(* IEC 61131-3 sources: Intern_HiERN_Testplattform_Hoplyt/Intern_HiERN_Testplattform_PLC, 10 files *)

(* ---- GlobalVariables.gvl ---- *)
VAR_GLOBAL
	MFC_INSTANCE : MFC_BHFF;

	MFC_CONTROLLER: FB_Bronkhorst_FFDevice_RTU;

	CORIFLOW_INSTANCE : BH_DeviceSingle;
	CORIFLOW_CONTROLLER: FB_Bronkhorst_SingleDevice;

	ELPRESS_INSTANCE : BH_DeviceSingle;
	ELPRESS_CONTROLLER: FB_Bronkhorst_SingleDevice;

	TESTCASE: TESTCASE;

	(* HW *)
	Read_SV_flow : REAL;
	Read_AV_flow : REAL;
	Read_unit_flow : STRING;
	Read_alarm_info_flow : SINT;

	Read_SV_p_up : REAL;
	Read_AV_p_up : REAL;
	Read_unit_p_up : STRING;
	Read_alarm_info_p_up : SINT;

	Read_SV_p_down : REAL;
	Read_AV_p_down : REAL;
	Read_unit_p_down : STRING;
	Read_alarm_info_p_down : SINT;

	Read_temperature: REAL;
	Read_density: REAL;

	Read_UserTag : STRING;
	Read_FluidName: STRING;
	Read_SN : STRING;
	Read_status : SINT;
	Read_AlarmMode : SINT;
	Read_ControlMode : SINT;
	Read_ControlFunction : SINT;

	Write_SVreq_flow : REAL;
	Write_SVreq_p_up : REAL;
	Write_SVreq_p_down : REAL;
	Write_ControlMode : SINT;
	Write_ControlFunction : SINT;
	Write_UserTag : STRING;
	Write_Reset_to_device : SINT;
	Write_Reset_Alarm_Enable : SINT;

	(* Huber Piccolo Thermostat & Debug Data Structures *)
	thermostat_1 : Thermostat;
	ser_debug    : serial_debug;
END_VAR

(* ---- FB_BlinkTakt.st ---- *)
(******************************************************************************
Description: Blink Takt Generator

Generates a symmetrical blinking signal using internal TON and TP timers.
The blink period is defined via the input time and split into equal ON/OFF phases.
A rising edge detector ensures clean toggling of the blink signal.

Input:
  - IN_period : TIME
      Total blink period (e.g. T#1s for 1 Hz blink).
      The signal will be HIGH for half the period and LOW for the other half.

Output:
  - Out_BlinkTakt : BOOL
      The generated blinking signal with a 50% duty cycle.

Internal:
  - HalfTime : TIME
      Half of the total blink period (IN_period / 2).
	  Defines both the ON and OFF duration to achieve a symmetrical 50 % duty cycle.
  - BlinkTON : TON
      On-delay timer used as the periodic time base.
	  The timer measures each half-period and signals its completion via Q, upon which the blink state is toggled and the timer cycle restarts.
  - BlinkState : BOOL
	  Internal state variable holding the current blink state.
	  The value is toggled once every half-period when BlinkTON.Q becomes TRUE and directly drives the output Out_BlinkTakt.

Return: Output variable `Out_BlinkTakt` provides the blinking signal.
******************************************************************************)

FUNCTION_BLOCK FB_BlinkTakt
VAR_INPUT
IN_period : TIME;
END_VAR

VAR_OUTPUT
Out_BlinkTakt : BOOL;
END_VAR

VAR

    HalfTime : TIME;
    BlinkTON : TON;
    BlinkState : BOOL := FALSE;

END_VAR

HalfTime := IN_period / 2;

BlinkTON(IN := NOT BlinkTON.Q, PT := HalfTime);

IF BlinkTON.Q THEN
    BlinkState := NOT BlinkState;
END_IF;

Out_BlinkTakt := BlinkState;

END_FUNCTION_BLOCK

(* ---- FB_Bronkhorst_FFDevice_RTU.st ---- *)
FUNCTION_BLOCK FB_Bronkhorst_FFDevice_RTU
VAR_INPUT
	Input_DeviceInstance: MFC_BHFF;

	Input_flow: FF_ProcessValue;
	Input_p_up: FF_ProcessValue;
	Input_p_down: FF_ProcessValue;

	Input_UserTag : STRING;
	Input_FluidName : STRING;
	Input_SN : STRING;
	Input_status : SINT;
	Input_AlarmMode : SINT;
	Input_ControlMode : SINT := 23; (*23: CONTROLMODE_DEACTIVATED*)
	Input_ControlFunction : SINT;
	Input_AV_Timeout : TIME := T#300s;
	Input_SV_Accept_Timeout: TIME := T#10s;

END_VAR

VAR_OUTPUT

	Output_SVreq_flow : REAL;
	Output_SVreq_p_up : REAL;
	Output_SVreq_p_down : REAL;
	Output_ControlMode : SINT;
	Output_ControlFunction : SINT;
	Output_Reset_to_device : SINT;
	Output_UserTag : STRING;
	Output_ErrorState : state_device_error := DEV_ERR_NONE;
	Output_DeviceInstance : MFC_BHFF;

END_VAR

VAR_IN_OUT

END_VAR

VAR
	state			: state_device := DV_INIT;
	state_next		: state_device := DV_INIT;
    state_prev      : state_device := DV_INIT;
    StateEntry		: BOOL;

    (* ==== Initialisierung ==== *)

    t_init_timeout   : TON;
    init_timeout     : TIME := T#5s;

    sn_valid         : BOOL;
    msg_str			 : STRING(255) := 'Device disabled.';

    req_reset		 : BOOL := FALSE;

	Input_alarm_info_flow : ARRAY [1..8] OF BOOL;
	Input_alarm_info_p_up : ARRAY [1..8] OF BOOL;
	Input_alarm_info_p_down : ARRAY [1..8] OF BOOL;

	Input_p_up_SV_mbarg: REAL; (* mbar(g) *)
	Input_p_up_AV_mbarg: REAL; (* mbar(a) *)
	Input_p_up_unit_mbarg: STRING := 'mbar (g)'; (* mbar (g) *)

	Input_p_down_SV_mbarg: REAL; (* mbar(g) *)
	Input_p_down_AV_mbarg: REAL; (* mbar(g) *)
	Input_p_down_unit_mbarg: STRING := 'mbar (g)'; (* mbar(g) *)

	FLAG_Alarm: BOOL := FALSE;
	FLAG_Warning: BOOL := FALSE;

    (* ==== Konfigurations-Latches ==== *)
    cfg_function_req : SINT;
    cfg_function_act : SINT;

    cfg_mode_req     : SINT;
    cfg_mode_act     : SINT;
    setpoint_mode_allowed : BOOL;

    cfg_pending      : BOOL;   (* TRUE sobald Funktion ODER Mode geändert wurde *)

    (* ==== SV-Latches ==== *)
    sv_req : FF_SV_LATCH;

	activePrimary : BH_ActiveChannel;
	activeSecondary : BH_ActiveChannel;
	secondaryChannelActive : BOOL;

	sv_rejected		 : BOOL;
	sv_changed		 : BOOL;
	sv_outofrange	 : BOOL;
    sv_pending       : BOOL;
    sv_applied		 : BOOL;
    sv_reached		 : BOOL;
    sv_maintained	 : BOOL;
    sv_accepted      : BOOL;   (* Gerät hat SV übernommen *)
    sv_active		 : BOOL;

   	SV_lower_range_limit : REAL;
	SV_upper_range_limit : REAL;
	AV_lower_range_limit : REAL;
	AV_upper_range_limit : REAL;
	SV_tolerance : REAL := 1.0; (* Fallback-Wert - Einstellung über User.Settings*)
	SV_in_range : BOOL := FALSE;
	AV_in_range : BOOL := FALSE;

    t_sv_accept   		: TON;
    t_av_timeout		: TON;
    t_av_NOTmaintained	: TON;

	(* ==== User Messages ==== *)
	prefix	: STRING;
	cf_str 	: STRING;
	cm_str	: STRING;
	sv_str	: STRING;
	unit_str: STRING;
	dev_status_str: STRING(255);
	err_msg	: STRING(255);
	warning_detail_str : STRING(255);

    (* ==== Magic Numbers ==== *)
	CONTROLMODE_DEACTIVATED : SINT := 23;
   	P_MAX_BAR : REAL := 3000.0; (* mbar (g)*)

	(* ==== Labels ==== *)
	alarm_lable : STRING := 'Alarm: ';
	error_lable : STRING := 'Error: ';
	warning_lable : STRING := 'Warning: ';
	notification_lable : STRING := 'Info: ';

	k : INT;

END_VAR

(* Eingangsdaten *)
Output_DeviceInstance := Input_DeviceInstance;
ACT_ProcessAlarmInfo_Input;
ACT_pInput_bara_to_mbarg;

(* User Requests *)
ACT_Latch_ControlFunction;
ACT_Latch_ControlMode;
ACT_Latch_SVreq;

(* Diagnose *)
ACT_Map_AlarmInfo;
ACT_AlarmInfo_wo_text;
ACT_Status_wo_text;

ACT_SelectActiveChannel;

(* STATE MACHINE *)
state_prev := state;
state := state_next;
StateEntry := state <> state_prev;

CASE state OF

	DV_INIT:
			ACT_Init;
			setpoint_mode_allowed := FALSE;

	DV_DISABLED:
			setpoint_mode_allowed := FALSE;
			IF Input_DeviceInstance.enable THEN
				state_next := DV_IDLE;
			ELSE
				ACT_Central_SVreq_Discard;
			END_IF

	DV_IDLE:
			IF StateEntry THEN
				ACT_Central_SVreq_Discard;
			END_IF

			(* === State neu festlegen === *)
			IF cfg_pending OR sv_pending THEN
				state_next := DV_SETTING_REQ;
			END_IF
			;

	DV_SETTING_REQ:
			ACT_Commit_Config;

			IF sv_pending OR sv_applied THEN
				ACT_Handle_SV;
			END_IF

			(* === State neu festlegen === *)
	        IF NOT cfg_pending AND NOT sv_pending AND NOT sv_applied AND NOT sv_accepted THEN
	            state_next := DV_IDLE;
	        ELSIF sv_accepted THEN
	            state_next := DV_CONTROLLING;
	        ELSIF t_sv_accept.Q THEN
				Output_ErrorState := DEV_ERR_SV_ACCEPT_TIMEOUT;
			    state_next := DV_ERROR;
	        END_IF
			;
	DV_CONTROLLING:
			IF cfg_pending THEN
				state_next := DV_IDLE;
			ELSIF sv_pending THEN
				state_next := DV_SETTING_REQ;
			ELSIF NOT sv_active THEN
	            state_next := DV_IDLE;
	        ELSIF sv_reached THEN
	            state_next := DV_SETTLED;
	        ELSIF t_av_timeout.Q THEN
            	Output_ErrorState := DEV_ERR_AV_Reach_TIMEOUT;
                state_next := DV_ERROR;
            ELSE
            	ACT_Controlling;
			END_IF
			;
	DV_SETTLED:
			IF cfg_pending THEN
				state_next := DV_IDLE;
			ELSIF sv_pending THEN
				state_next := DV_SETTING_REQ;
			ELSIF NOT sv_active THEN
	            state_next := DV_IDLE;
	        ELSIF t_av_NOTmaintained.Q THEN
            	state_next := DV_ERROR;
            	Output_ErrorState := DEV_ERR_AV_Maintain_TIMEOUT;
            ELSE
            	ACT_Settled;
			END_IF

			;
	DV_ERROR:
			ACT_Latch_Reset;
			setpoint_mode_allowed := FALSE;
			IF req_reset THEN

				ACT_Reset_BH_Device;
				state_next := DV_IDLE;
				req_reset := FALSE;

				Output_ErrorState := DEV_ERR_NONE;
			END_IF
END_CASE

(* GLOBAL STATE TRANSITIONS *)
IF FLAG_Alarm THEN
	state_next := DV_ERROR;

ELSIF NOT Input_DeviceInstance.enable THEN
	state_next := DV_DISABLED;
END_IF

(* Outputs *)
ACT_Output_To_Device_And_User;
ACT_Build_StatusMessage;

END_FUNCTION_BLOCK

ACTIONS
	ACTION ACT_Init

		IF StateEntry THEN
	    (* Timeout starten *)
	   		t_init_timeout(IN := TRUE, PT := init_timeout);
	    END_IF

	    (* Seriennummer vom Gerät lesen *)
	    Output_DeviceInstance.serialnumber := Input_SN;

	    (* Plausibilitätsprüfung *)
	    sn_valid := (LEN(Input_SN) >= 4) AND (Input_SN <> '0000');

	    IF sn_valid THEN
	        (* Verbindung erfolgreich *)
	        t_init_timeout(IN := FALSE);
	        Output_DeviceInstance.status_msg :=  CONCAT('Device connection established. SN=',Input_SN);

			(* Erstmaligen Status abrufen *)
		    cfg_pending := TRUE;

		    ACT_cfg_function_feedback;
		    ACT_cfg_mode_feedback;

		    Output_ErrorState := DEV_ERR_NONE;
		    state_next := DV_IDLE;
	    END_IF

	    (* Timeout abgelaufen -> Fehler *)
	    IF t_init_timeout.Q THEN
			Output_ErrorState := DEV_ERR_INIT;
	        Output_DeviceInstance.status_msg := 'ERROR: Device connection timeout – no valid serial number';
	        state_next := DV_ERROR;
	    END_IF

	END_ACTION

	ACTION ACT_pInput_bara_to_mbarg
		Input_p_up_SV_mbarg := Input_p_up.SV*1000-1000; (* mbar(g) *)
		Input_p_up_AV_mbarg := Input_p_up.AV*1000-1000; (* mbar(a) *)

		Input_p_down_SV_mbarg := Input_p_down.SV*1000-1000; (* mbar(g) *)
		Input_p_down_AV_mbarg := Input_p_down.AV*1000-1000; (* mbar(g) *)
	END_ACTION

	ACTION ACT_Latch_Reset

		(* ERROR Reset *)

		req_reset := Input_DeviceInstance.reset;
		Input_DeviceInstance.reset := FALSE;
		Output_DeviceInstance.reset := FALSE;
	END_ACTION

	ACTION ACT_Latch_ControlFunction
	    (* ControlFunction *)
	    IF Input_DeviceInstance.control_function_req <> Input_ControlFunction THEN
	        cfg_function_req := Input_DeviceInstance.control_function_req;
	        cfg_pending := TRUE;
	    END_IF
	    cfg_function_act := Input_ControlFunction;

	    IF cfg_pending THEN
	    	ACT_Central_SVreq_Discard;
	    END_IF
	END_ACTION

	ACTION ACT_Latch_ControlMode
	    (* ControlMode *)
	    IF Input_DeviceInstance.control_mode_req <> Input_ControlMode THEN
	        cfg_mode_req := Input_DeviceInstance.control_mode_req;
	        cfg_pending := TRUE;
	    END_IF
	    cfg_mode_act := Input_ControlMode;

	    setpoint_mode_allowed := (cfg_mode_act = 0);   (* 0 = BUS/RS232 *)

	    IF NOT setpoint_mode_allowed THEN
	    	ACT_Central_SVreq_Discard;
	    END_IF
	END_ACTION

	ACTION ACT_Latch_SVreq
	    (* SV Requests *)
	    IF NOT cfg_pending AND setpoint_mode_allowed THEN

	    sv_changed := FALSE;

	    	CASE cfg_function_act OF
		    0:
		    	sv_changed := ABS(Input_DeviceInstance.SV_flow_req - Input_flow.SV) >= 0.001;

				IF sv_changed THEN
		            sv_req.Flow := Input_DeviceInstance.SV_flow_req;
		        END_IF
			1:
		        sv_changed := ABS(Input_DeviceInstance.SV_p_up_req - Input_p_up_SV_mbarg) >= 0.001;

				IF sv_changed THEN
		            sv_req.PUp := Input_DeviceInstance.SV_p_up_req;
		        END_IF
			2:
		        sv_changed := ABS(Input_DeviceInstance.SV_p_down_req - Input_p_down_SV_mbarg) >= 0.001;

				IF sv_changed THEN
		            sv_req.PDown := Input_DeviceInstance.SV_p_down_req;
				END_IF
			4:
				sv_changed := ABS(Input_DeviceInstance.SV_p_down_req - Input_p_down_SV_mbarg) >= 0.001 OR
					ABS(Input_DeviceInstance.SV_flow_req - Input_flow.SV) >= 0.001;

				IF sv_changed THEN
		            sv_req.PDown := Input_DeviceInstance.SV_p_down_req;
		            sv_req.Flow := Input_DeviceInstance.SV_flow_req;
		        END_IF
		    END_CASE

		    IF sv_changed THEN
				ACT_Reset_SV_Lifecycle;	(* Lebenszyklus neu starten *)
	            sv_pending := TRUE;
	        END_IF

	    END_IF

	END_ACTION

	ACTION ACT_Reset_SV_Lifecycle
		sv_rejected := FALSE;
	    sv_applied  := FALSE;
	    sv_accepted := FALSE;
	    sv_reached  := FALSE;
	    sv_maintained := FALSE;

	    t_sv_accept(IN := FALSE);
		t_av_timeout(IN := FALSE);
		t_av_NOTmaintained(IN := FALSE);

	END_ACTION

	ACTION ACT_Controlling
			(* === CONTROLLING: Überwachung === *)

	        (* Timeout *)
	        CASE cfg_function_act OF
	        0..2:
	        	t_av_timeout(IN := NOT sv_reached, PT := Input_AV_Timeout);
	        4:
	        	t_av_timeout(IN := NOT sv_reached, PT := T#300s);
	        END_CASE

	        IF t_av_timeout.Q THEN
	        	RETURN;
	        END_IF

	        (* Toleranzprüfung *)
	        AV_lower_range_limit := activePrimary.SVreq * (100.0-(SV_tolerance*0.5))/100.0;
			AV_upper_range_limit := activePrimary.SVreq * (100.0+(SV_tolerance*0.5))/100.0;

			AV_in_range := INRANGE(AV_lower_range_limit,activePrimary.AV,AV_upper_range_limit);

	        IF AV_in_range THEN
	            sv_reached := TRUE;
	        ELSE
	        	sv_reached := FALSE;
	        END_IF

	END_ACTION

	ACTION ACT_Settled
			(* Timeout *)
	    	t_av_NOTmaintained(IN := NOT sv_maintained, PT := T#10s); (* Variabel über User !!*)

	        (* Rückfall, falls Wert wieder wegdriftet *)
	        AV_lower_range_limit := activePrimary.SVreq * (100.0-(SV_tolerance*1))/100.0;
			AV_upper_range_limit := activePrimary.SVreq * (100.0+(SV_tolerance*1))/100.0;

			AV_in_range := INRANGE(AV_lower_range_limit,activePrimary.AV,AV_upper_range_limit);
	        IF AV_in_range THEN
	        	sv_maintained := TRUE;
	        ELSE
	        	sv_maintained := FALSE;
	        END_IF
	END_ACTION

	ACTION ACT_Central_SVreq_Discard

        sv_pending := FALSE;

        (* SV-Latches zurücksetzen *)
		sv_req.Flow   := 0.0;
	    sv_req.PUp   := 0.0;
	    sv_req.PDown := 0.0;

        (* Lebenszyklus vollständig zurücksetzen *)
        ACT_Reset_SV_Lifecycle;

        (* Rückmeldung an User *)
        Output_DeviceInstance.SV_flow_req   := 0.0;
        Output_DeviceInstance.SV_p_up_req   := 0.0;
        Output_DeviceInstance.SV_p_down_req := 0.0;

		(* Device Reset zurücksetzten *)
		Output_Reset_to_device := 0;
	END_ACTION

	ACTION ACT_cfg_function_feedback
		CASE cfg_function_act OF
	        0: cf_str := ': Flow';
	        1: cf_str := ': Upstream pressure';
	        2: cf_str := ': Downstream pressure';
	        4: cf_str := ': Downstream pressure with flow limit';
	    ELSE
            cf_str := ' - undefined';
        END_CASE
	END_ACTION

	ACTION ACT_cfg_mode_feedback
		CASE cfg_mode_act OF
			0: cm_str := 'BUS/RS232';
			1: cm_str := 'Analog input';
			2: cm_str := 'FLOW-BUS slave';
			3: cm_str := 'Valve close';
			4: cm_str := 'Controller idle';
			5: cm_str := 'Testing mode';
			6: cm_str := 'Tuning mode';
			7: cm_str := 'Setpoint 100%';
			8: cm_str := 'Valve fully open';
			9: cm_str := 'Calibration mode';
			10: cm_str := 'Analog slave';
			12: cm_str := 'setpoint 0%';
			13: cm_str := 'FLOW-BUS analog slave';
			18: cm_str := 'RS232';
			20: cm_str := 'valve steering (valve = setpoint)';
			21: cm_str := 'analog valve steering(valve = analog input)';
			22: cm_str := 'valve safe state';
		ELSE
            cm_str := ' - undefined';
		END_CASE
	END_ACTION

	ACTION ACT_SelectActiveChannel

		secondaryChannelActive := FALSE;

		CASE cfg_function_act OF

		0: (* Flow *)
			activePrimary.SVreq := sv_req.Flow;
			activePrimary.AV := Input_flow.AV;
			activePrimary.DeviceSV := Input_flow.SV;
			activePrimary.Unit := Input_flow.Unit;
			activePrimary.SV_Min := Input_DeviceInstance.lower_limit;
			activePrimary.SV_Max := Input_DeviceInstance.upper_limit;
		1: (* Upstream Pressure *)
			activePrimary.SVreq := sv_req.PUp;
			activePrimary.AV := Input_p_up_AV_mbarg;
			activePrimary.DeviceSV := Input_p_up_SV_mbarg;
			activePrimary.Unit := Input_p_up_unit_mbarg;
			activePrimary.SV_Min := 0.0;
			activePrimary.SV_Max := P_MAX_BAR;
		2: (* Downstream Pressure *)
			activePrimary.SVreq := sv_req.PDown;
			activePrimary.AV := Input_p_down_AV_mbarg;
			activePrimary.DeviceSV := Input_p_down_SV_mbarg;
			activePrimary.Unit := Input_p_down_unit_mbarg;
			activePrimary.SV_Min := 0.0;
			activePrimary.SV_Max := P_MAX_BAR;
		4: (* Downstream Pressure w flow limit *)
			activePrimary.SVreq := sv_req.PDown;
			activePrimary.AV := Input_p_down_AV_mbarg;
			activePrimary.DeviceSV := Input_p_down_SV_mbarg;
			activePrimary.Unit := Input_p_down_unit_mbarg;
			activePrimary.SV_Min := 0.0;
			activePrimary.SV_Max := P_MAX_BAR;

			secondaryChannelActive := TRUE;
			activeSecondary.SVreq := sv_req.Flow;
			activeSecondary.AV := Input_flow.AV;
			activeSecondary.DeviceSV := Input_flow.SV;
			activeSecondary.Unit := Input_flow.Unit;
			activeSecondary.SV_Min := Input_DeviceInstance.lower_limit;
			activeSecondary.SV_Max := Input_DeviceInstance.upper_limit;

		END_CASE

		sv_active := (activePrimary.SVreq <> 0.0);
	END_ACTION

	ACTION ACT_Commit_Config

	    IF cfg_pending THEN

	        (* === Commit ControlFunction === *)
	        Output_ControlFunction := cfg_function_req;

	        IF Input_ControlFunction = cfg_function_req THEN
		       ACT_cfg_function_feedback;
	        END_IF

			 (* === Commit ControlMode === *)
	        Output_ControlMode := cfg_mode_req;

			IF Input_ControlMode = cfg_mode_req THEN
		        ACT_cfg_mode_feedback;
	        END_IF

			IF  Input_ControlMode = cfg_mode_req AND Input_ControlFunction = cfg_function_req THEN
		        cfg_pending := FALSE;
	        END_IF

	    END_IF

	END_ACTION

	ACTION ACT_Handle_SV

		IF NOT setpoint_mode_allowed THEN
		    sv_rejected := TRUE;
		    RETURN;
		END_IF

	    (* Nur relevante States - nötig? *)
	    IF (state <> DV_SETTING_REQ) AND
	       (state <> DV_CONTROLLING) AND
	       (state <> DV_SETTLED) THEN
	        sv_rejected := TRUE;
	        RETURN;
	    END_IF

	    (* Keine Arbeit bei Config-Wechsel *)
	    IF cfg_pending THEN
	    	sv_rejected := TRUE;
	        RETURN;
	    END_IF

		sv_str := CONCAT(REAL_TO_STRING(activePrimary.SVreq),activePrimary.Unit);

	    IF secondaryChannelActive THEN
			sv_str := CONCAT(sv_str,' (Flow limit ');
			sv_str := CONCAT(sv_str,REAL_TO_STRING(activeSecondary.SVreq));
			sv_str := CONCAT(sv_str,' ');
			sv_str := CONCAT(sv_str,activeSecondary.Unit);
			sv_str := CONCAT(sv_str,')');
		END_IF

		IF NOT sv_applied THEN

	        (* Bereich prüfen *)
			SV_in_range := INRANGE(activePrimary.SV_Min, activePrimary.SVreq, activePrimary.SV_Max);

			IF NOT SV_in_range THEN
			    (* === Ungültigen User-Sollwert zurückweisen === *)

			    sv_pending := FALSE;

				IF activePrimary.SVreq < activePrimary.SV_Min OR activePrimary.SVreq > activePrimary.SV_Max THEN
				    (* User-SV auf aktuell gültigen Sollwert zurücksetzen *)
				    ACT_Restore_UserSetpoints;

				    (* Optional: Statusmeldung *)
				    sv_outofrange := TRUE;
					sv_rejected := TRUE;

				    RETURN;
				  END_IF
			END_IF

			sv_outofrange := FALSE;
	        sv_applied := TRUE;
	        sv_pending := FALSE;
		END_IF

		(* Prüfen, ob Gerät SV übernommen hat *)
		IF sv_applied AND NOT sv_accepted THEN
			(* Akzeptanz-Timer starten *)
		    t_sv_accept(IN := TRUE, PT := Input_SV_Accept_Timeout);

		    IF NOT secondaryChannelActive THEN

				IF activePrimary.SVreq = activePrimary.DeviceSV THEN
					sv_accepted := TRUE;
				END_IF

			ELSE

				IF ABS(activePrimary.SVreq - activePrimary.DeviceSV)<= activePrimary.SVreq * 0.01 AND
					activeSecondary.SVreq = activeSecondary.DeviceSV THEN
					sv_accepted := TRUE;
				END_IF

			END_IF

		END_IF

	END_ACTION

	ACTION ACT_Restore_UserSetpoints
		 Output_DeviceInstance.SV_flow_req   := sv_req.Flow;
		 Output_DeviceInstance.SV_p_up_req   := sv_req.PUp;
		 Output_DeviceInstance.SV_p_down_req := sv_req.PDown;
	END_ACTION

	ACTION ACT_Output_To_Device_And_User

	    (* ================================================= *)
	    (* Default: keine Sollwerte an das Gerät             *)
	    (* ================================================= *)
	    Output_SVreq_flow   := 0.0;
	    Output_SVreq_p_up   := 0.0;
	    Output_SVreq_p_down := 0.0;

	    (* ================================================= *)
	    (* Sollwert nur ausgeben, wenn er gültig angewandt    *)
	    (* ================================================= *)
	    IF sv_applied AND
	       (state = DV_SETTING_REQ OR state = DV_CONTROLLING OR state = DV_SETTLED) THEN

	        CASE cfg_function_act OF

	            0:  (* Flow *)
	            	IF sv_req.Flow > 0 THEN
	                	Output_SVreq_flow := sv_req.Flow;
	                END_IF

	            1:  (* Upstream pressure *)
	                Output_SVreq_p_up := sv_req.PUp/1000+1; (* Umrechnung von mbar (g) zu bar (a) *)

	            2:  (* Downstream pressure *)
	                Output_SVreq_p_down := sv_req.PDown/1000+1; (* Umrechnung von mbar (g) zu bar (a) *)

	            4:  (* Downstream pressure with flow limit *)
	                Output_SVreq_p_down := sv_req.PDown/1000+1; (* Umrechnung von mbar (g) zu bar (a) *)
	                Output_SVreq_flow   := sv_req.Flow;

	        END_CASE
	    END_IF

	    (* ================================================= *)
	    (* Status an User                                    *)
	    (* ================================================= *)
		ACT_ReadAV;

	    Output_DeviceInstance.control_function := cfg_function_act;
	    Output_DeviceInstance.control_mode     := cfg_mode_act;
		Output_DeviceInstance.control_function_req := cfg_function_req;
	    Output_DeviceInstance.control_mode_req     := cfg_mode_req;

		Output_DeviceInstance.state := state;
		Output_DeviceInstance.enable := Input_DeviceInstance.enable;
		Output_DeviceInstance.SVaccepted := sv_accepted;
		Output_DeviceInstance.SVrejected := sv_rejected;
		Output_DeviceInstance.SVreached := sv_reached;
	    Output_DeviceInstance.SV_flow_req := sv_req.Flow;
	    Output_DeviceInstance.SV_flow := Input_flow.SV;
		Output_DeviceInstance.SV_p_up_req := sv_req.PUp;
		Output_DeviceInstance.SV_p_up := Input_p_up_SV_mbarg;
		Output_DeviceInstance.SV_p_down_req := sv_req.PDown;
		Output_DeviceInstance.SV_p_down := Input_p_down_SV_mbarg;

	END_ACTION

	ACTION ACT_Map_AlarmInfo

	    CASE cfg_function_act OF
	        0:  Output_DeviceInstance.alarm_info := Input_alarm_info_flow;
	        1:  Output_DeviceInstance.alarm_info := Input_alarm_info_p_up;
	        2,4: Output_DeviceInstance.alarm_info := Input_alarm_info_p_down;
	    END_CASE

	END_ACTION

	ACTION ACT_ReadAV
		Output_DeviceInstance.media := Input_FluidName;
		IF Input_flow.AV > Input_DeviceInstance.upper_limit/500 THEN
			Output_DeviceInstance.AV_flow := Input_flow.AV;
		ELSE Output_DeviceInstance.AV_flow := 0;
		END_IF;
		Output_DeviceInstance.unit_flow := Input_flow.Unit;
		Output_DeviceInstance.AV_p_up := Input_p_up_AV_mbarg;
		Output_DeviceInstance.unit_p := Input_p_up.Unit;
		Output_DeviceInstance.AV_p_down := Input_p_down_AV_mbarg;
		Output_DeviceInstance.unit_p := Input_p_down.Unit;
		Output_DeviceInstance.serialnumber := Input_SN;
		Output_DeviceInstance.name := Input_UserTag;
	END_ACTION

	ACTION ACT_ProcessAlarmInfo_Input

		Input_alarm_info_flow := BH_AlarmBitTOAlarmArray(Input_flow.AlarmInfo);
		Input_alarm_info_p_up := BH_AlarmBitTOAlarmArray(Input_p_up.AlarmInfo);
		Input_alarm_info_p_down := BH_AlarmBitTOAlarmArray(Input_p_down.AlarmInfo);

	END_ACTION

	ACTION ACT_AlarmInfo_wo_text

	    FLAG_Alarm := FALSE;
	    FLAG_Warning := FALSE;

		warning_detail_str := '';

	    FOR k := 1 TO 8 DO
	        IF Output_DeviceInstance.alarm_info[k] THEN

	            CASE k OF
	                1: (* Alarm *)
	                    FLAG_Alarm := TRUE;

	                2: (* Warning *)
	                    FLAG_Warning := TRUE;

	                3: (* Sensor < min *)
	                    FLAG_Warning := TRUE;
	                    warning_detail_str := CONCAT(warning_detail_str,'Sensor below minimum limit; ');

	                4: (* Sensor > max *)
	                    FLAG_Warning := TRUE;
	                    warning_detail_str := CONCAT(warning_detail_str,'Sensor above maximum limit; ');

	                5: (* Batch counter *)
	                    FLAG_Warning := TRUE;
	                    warning_detail_str := CONCAT(warning_detail_str,'Batch counter limit reached; ');

	                6: (* Power-up / deviation *)
	                    FLAG_Warning := TRUE;
	                    warning_detail_str := CONCAT(warning_detail_str,'Power-up alarm; ');

	                7: (* Communication *)
	                    FLAG_Alarm := TRUE;
	                    Output_ErrorState := DEV_ERR_COMMUNICATION;
	                8: (* Hardware *)
	                    FLAG_Alarm := TRUE;
	                    Output_ErrorState := DEV_ERR_HARDWARE;

	            END_CASE
	        END_IF
	    END_FOR

	    Output_DeviceInstance.warning := FLAG_Warning;
	    Output_DeviceInstance.alarm   := FLAG_Alarm;

	END_ACTION

	ACTION ACT_Status_wo_text

        Output_DeviceInstance.status := Input_status;

        (* Default zurücksetzen *)
        (* Wichtig: nicht alarm/warning global löschen! *)

        CASE Input_status OF

            0: (* Normal operation *)
                ;(* nichts setzen *)

            1: (* Maintenance required *)
                Output_DeviceInstance.warning := TRUE;

            2: (* Out of specification *)
                Output_DeviceInstance.warning := TRUE;

            4: (* Check function *)
                Output_DeviceInstance.warning := TRUE;

            8: (* Device failure *)
                Output_DeviceInstance.alarm := TRUE;
                FLAG_Alarm := TRUE;
                Output_ErrorState := DEV_ERR_DEVICE_FAILURE;

            ELSE
                (* unbekannter Status *)
                Output_DeviceInstance.warning := TRUE;

        END_CASE

	END_ACTION

	ACTION ACT_Name

		IF Input_UserTag <> Input_DeviceInstance.name THEN
			Output_UserTag := Input_DeviceInstance.name;;
			Output_DeviceInstance.name := Input_DeviceInstance.name;
		END_IF

	END_ACTION

	ACTION ACT_Build_StatusMessage

	    Output_DeviceInstance.status_msg := '';

	    (* === Priority Prefix === *)
	    IF state = DV_INIT THEN
	        Output_DeviceInstance.status_msg :=
	            CONCAT(notification_lable, 'Initializing device...');
	        RETURN;
	    END_IF

    	CASE Output_ErrorState OF

    		DEV_ERR_NONE: err_msg := '';

    		DEV_ERR_INIT: err_msg := 'Initialization timeout';

    		DEV_ERR_SV_ACCEPT_TIMEOUT: err_msg:= 'Set Value not accepted - TIMEOUT';

    		DEV_ERR_AV_Reach_TIMEOUT: err_msg:= 'Actual Value not in tolerance - TIMEOUT';

    		DEV_ERR_AV_Maintain_TIMEOUT: err_msg:= 'Actual Value not maintained - TIMEOUT';

    		DEV_ERR_COMMUNICATION: err_msg := 'Communication error';

    		DEV_ERR_HARDWARE: err_msg := 'Hardware alarm';

    		DEV_ERR_DEVICE_FAILURE: err_msg := 'Device failure';

    	END_CASE

		IF sv_rejected THEN
			Output_DeviceInstance.warning := TRUE;
			IF warning_detail_str <> '' THEN
				warning_detail_str :=CONCAT(warning_detail_str,', Setpoint rejected - ');
			ELSE
				warning_detail_str := 'Setpoint rejected - ';
			END_IF

			IF NOT setpoint_mode_allowed THEN
				warning_detail_str :=CONCAT(warning_detail_str,'no Setpoint allowed.');
			ELSIF cfg_pending THEN
				warning_detail_str :=CONCAT(warning_detail_str,'HW-Config pending.');
			ELSIF sv_outofrange THEN
				warning_detail_str :=CONCAT(warning_detail_str,'Setpoint out of range.');
			END_IF

		END_IF

	    IF Output_DeviceInstance.alarm THEN
	        prefix := alarm_lable;
	    ELSIF Output_DeviceInstance.warning THEN
	        prefix := warning_lable;
	    ELSE
	        prefix := notification_lable;
	    END_IF

	    Output_DeviceInstance.status_msg := prefix;

	    (* === ControlFunction / ControlMode === *)
	    Output_DeviceInstance.status_msg :=
	        CONCAT(Output_DeviceInstance.status_msg,'CF=');
	    Output_DeviceInstance.status_msg :=
	        CONCAT(Output_DeviceInstance.status_msg,cf_str);

		Output_DeviceInstance.status_msg :=
	        CONCAT(Output_DeviceInstance.status_msg,', CM=');
	    Output_DeviceInstance.status_msg :=
	        CONCAT(Output_DeviceInstance.status_msg,cm_str);

	    (* === Setpoint === *)
	    IF sv_applied THEN
	        Output_DeviceInstance.status_msg :=
		        CONCAT(Output_DeviceInstance.status_msg,', SV=');
		    Output_DeviceInstance.status_msg :=
		        CONCAT(Output_DeviceInstance.status_msg,sv_str);
	    END_IF

	    (* === State-dependent text === *)
	    CASE state OF
	        DV_IDLE:
	            msg_str := ' (Idle)';
	        DV_SETTING_REQ:
	            IF sv_accepted THEN
	                msg_str := ' (Setpoint accepted)';
	            ELSE
	                msg_str := ' (Waiting for device to accept setpoint)';
	            END_IF
	        DV_CONTROLLING:
	            msg_str := ' (Controlling)';
	        DV_SETTLED:
	            msg_str := ' (Setpoint reached)';
	        DV_DISABLED:
	            msg_str := ' (Disabled)';
	    ELSE
	        msg_str := '';
	    END_CASE

	    CASE Output_DeviceInstance.status OF
		    0:
		        dev_status_str := 'Normal operation';

		    1:
		        dev_status_str := 'Maintenance required';

		    2:
		        dev_status_str := 'Out of specification';

		    4:
		        dev_status_str := 'Check function';

		    8:
		        dev_status_str := 'Device failure';

		ELSE
		    dev_status_str := 'Unknown device status';
		END_CASE

	    Output_DeviceInstance.status_msg :=
	        CONCAT(Output_DeviceInstance.status_msg, msg_str);

		Output_DeviceInstance.status_msg :=
	        CONCAT(Output_DeviceInstance.status_msg,' | Status: ');
	    Output_DeviceInstance.status_msg :=
	        CONCAT(Output_DeviceInstance.status_msg,dev_status_str);

		IF err_msg <> '' THEN
    		Output_DeviceInstance.status_msg := CONCAT(Output_DeviceInstance.status_msg,' | ');
    		Output_DeviceInstance.status_msg := CONCAT(Output_DeviceInstance.status_msg, error_lable);
        	Output_DeviceInstance.status_msg := CONCAT(Output_DeviceInstance.status_msg, err_msg);
	    END_IF

	    IF warning_detail_str <> '' THEN
	    	Output_DeviceInstance.status_msg := CONCAT(Output_DeviceInstance.status_msg,' | ');
	    	Output_DeviceInstance.status_msg := CONCAT(Output_DeviceInstance.status_msg,warning_detail_str);
	    END_IF
	END_ACTION

	ACTION ACT_Reset_BH_Device

		IF Input_DeviceInstance.alarm_reset_enable = 4 THEN
			Output_Reset_to_device := 2; (*reset alarm*)
			msg_str := ': Device reset triggered.';
		    Output_DeviceInstance.status_msg := CONCAT(notification_lable, Input_DeviceInstance.name);
		    Output_DeviceInstance.status_msg := CONCAT(Output_DeviceInstance.status_msg, msg_str);
		    Output_DeviceInstance.reset := FALSE;
		 ELSE
		 	msg_str := ': Device reset NOT available.';
		    Output_DeviceInstance.status_msg := CONCAT(warning_lable, Input_DeviceInstance.name);
		    Output_DeviceInstance.status_msg := CONCAT(Output_DeviceInstance.status_msg, msg_str);
		 END_IF

	END_ACTION

(*	ACTION ACT_Serialnumber_identification *)

(*		FOR i:= 1 TO 20 DO *)
(*			IF i=1 THEN *)
(*				string_var := ''; *)
(*			END_IF *)
(*			ascii_byte := Input_SN_from_device[i]; *)
(*			string_var := CONCAT(string_var, Util_Chr(ascii_byte)); *)
(*		END_FOR *)

(*	Output_DeviceInstance.serialnumber := string_var; *)

(*	Output_DeviceInstance.serialnumber := Input_SN; *)
(*	END_ACTION *)

END_ACTIONS

(* ---- FB_Bronkhorst_SingleDevice.st ---- *)
FUNCTION_BLOCK FB_Bronkhorst_SingleDevice
VAR_INPUT
	Input_DeviceInstance: BH_DeviceSingle;
	Input_DeviceType: BH_DeviceSingleType;

	Input: FF_ProcessValue;

	Input_temperature: REAL;
	Input_density: REAL;

	Input_UserTag: STRING;
	Input_FluidName: STRING;
	Input_SN : STRING;
	Input_status : SINT;
	Input_AlarmMode : SINT;
	Input_ControlMode: SINT := 23; (* 23 = deactivated *)
	Input_AV_Timeout : TIME := T#300s;
	Input_SV_Accept_Timeout: TIME := T#10s;

END_VAR

VAR_OUTPUT

	Output_SVreq : REAL;

	Output_ControlMode: SINT;
	Output_ControlFunction: SINT;
	Output_Reset_to_device : SINT;
	Output_Reset_Alarm_Enable : SINT := 0;
	Output_UserTag : STRING;
	Output_DeviceInstance : BH_DeviceSingle;
	Output_ErrorState : state_device_error := DEV_ERR_NONE;

END_VAR

VAR_IN_OUT
END_VAR

VAR
	state			: state_device := DV_INIT;
	state_next		: state_device := DV_INIT;
    state_prev      : state_device := DV_INIT;
    StateEntry		: BOOL;

    (* ==== Initialisierung ==== *)

    t_init_timeout   : TON;
    init_timeout     : TIME := T#5s;

    sn_valid         : BOOL;
    msg_str			 : STRING(255) := 'Device disabled.';

    req_reset		 : BOOL := FALSE;

	Input_alarm_info : ARRAY [1..8] OF BOOL;

	Input_p_SV_mbarg: REAL; (* mbar(g) *)
	Input_p_AV_mbarg: REAL; (* mbar(g) *)
	Input_p_unit_mbarg: STRING := 'mbar (g)'; (* mbar(g) *)

	FLAG_Alarm: BOOL := FALSE;
	FLAG_Warning: BOOL := FALSE;

    (* ==== Konfigurations-Latches ==== *)
    cfg_function_req : SINT;
    cfg_function_act : SINT;

    cfg_mode_req     : SINT;
    cfg_mode_act     : SINT;
    setpoint_mode_allowed : BOOL;

    cfg_pending      : BOOL;   (* TRUE sobald Funktion ODER Mode geändert wurde *)

    (* ==== SV-Latches ==== *)
    sv_req           : REAL;

	activePrimary    : BH_ActiveChannel;

	sv_rejected		 : BOOL;
	sv_rejected_latched : BOOL;
	sv_changed		 : BOOL;
	sv_outofrange	 : BOOL;
    sv_pending       : BOOL;
    sv_applied		 : BOOL;
    sv_reached		 : BOOL;
    sv_maintained	 : BOOL;
    sv_accepted      : BOOL;   (* Gerät hat SV übernommen *)
    sv_active		 : BOOL;

   	SV_lower_range_limit : REAL;
	SV_upper_range_limit : REAL;
	AV_lower_range_limit : REAL;
	AV_upper_range_limit : REAL;
	SV_tolerance : REAL := 1.0; (* Fallback-Wert - Einstellung über User.Settings*)
	SV_in_range : BOOL := FALSE;
	AV_in_range : BOOL := FALSE;

    t_sv_accept   		: TON;
    t_av_timeout		: TON;
    t_av_NOTmaintained	: TON;

	(* ==== User Messages ==== *)
	prefix	: STRING;
	dv_str 	: STRING;
	cm_str	: STRING;
	sv_str	: STRING;
	unit_str: STRING;
	dev_status_str: STRING(255);
	err_msg	: STRING(255);
	warning_detail_str : STRING(255);

    (* ==== Magic Numbers ==== *)
	CONTROLMODE_DEACTIVATED : SINT := 23;
   	P_MAX_BAR : REAL := 3000.0; (* mbar (g)*)

	(* ==== Labels ==== *)
	alarm_lable : STRING := 'Alarm: ';
	error_lable : STRING := 'Error: ';
	warning_lable : STRING := 'Warning: ';
	notification_lable : STRING := 'Info: ';

	k : INT;

END_VAR

(* Eingangsdaten *)
Output_DeviceInstance := Input_DeviceInstance;
ACT_ProcessAlarmInfo_Input;
ACT_pInput_bara_to_mbarg;

(* User Requests *)
ACT_Latch_ControlMode;
ACT_Latch_SVreq;

(* Diagnose *)
ACT_Map_AlarmInfo;
ACT_AlarmInfo_wo_text;
ACT_Status_wo_text;

ACT_SelectActiveChannel;

(* STATE MACHINE *)
state_prev := state;
state := state_next;
StateEntry := state <> state_prev;

CASE state OF

	DV_INIT:
			ACT_Init;
			setpoint_mode_allowed := FALSE;

	DV_DISABLED:
			setpoint_mode_allowed := FALSE;
			IF Input_DeviceInstance.enable THEN
				state_next := DV_IDLE;
			ELSE
				ACT_Central_SVreq_Discard;
			END_IF

	DV_IDLE:
			IF StateEntry THEN
				ACT_Central_SVreq_Discard;
			END_IF

			(* === State neu festlegen === *)
			IF cfg_pending OR sv_pending THEN
				state_next := DV_SETTING_REQ;
			END_IF
			;

	DV_SETTING_REQ:
			ACT_Commit_Config;

			IF sv_pending OR sv_applied THEN
				ACT_Handle_SV;
			END_IF

			(* === State neu festlegen === *)
	        IF NOT cfg_pending AND NOT sv_pending AND NOT sv_applied AND NOT sv_accepted THEN
	            state_next := DV_IDLE;
	        ELSIF sv_accepted THEN
	            state_next := DV_CONTROLLING;
	        ELSIF t_sv_accept.Q THEN
				Output_ErrorState := DEV_ERR_SV_ACCEPT_TIMEOUT;
			    state_next := DV_ERROR;
	        END_IF
			;
	DV_CONTROLLING:
			IF cfg_pending THEN
				state_next := DV_IDLE;
			ELSIF sv_pending THEN
				state_next := DV_SETTING_REQ;
			ELSIF NOT sv_active THEN
	            state_next := DV_IDLE;
	        ELSIF sv_reached THEN
	            state_next := DV_SETTLED;
	        ELSIF t_av_timeout.Q THEN
            	Output_ErrorState := DEV_ERR_AV_Reach_TIMEOUT;
                state_next := DV_ERROR;
            ELSE
            	ACT_Controlling;
			END_IF
			;
	DV_SETTLED:
			IF cfg_pending THEN
				state_next := DV_IDLE;
			ELSIF sv_pending THEN
				state_next := DV_SETTING_REQ;
			ELSIF NOT sv_active THEN
	            state_next := DV_IDLE;
	        ELSIF t_av_NOTmaintained.Q THEN
            	state_next := DV_ERROR;
            	Output_ErrorState := DEV_ERR_AV_Maintain_TIMEOUT;
            ELSE
            	ACT_Settled;
			END_IF

			;
	DV_ERROR:
			ACT_Latch_Reset;
			setpoint_mode_allowed := FALSE;
			IF req_reset THEN

				ACT_Reset_BH_Device;
				state_next := DV_IDLE;
				req_reset := FALSE;

				Output_ErrorState := DEV_ERR_NONE;
			END_IF
END_CASE

(* GLOBAL STATE TRANSITIONS *)
IF FLAG_Alarm THEN
	state_next := DV_ERROR;

ELSIF NOT sn_valid THEN
	state_next := DV_INIT;

ELSIF NOT Input_DeviceInstance.enable THEN
	state_next := DV_DISABLED;
END_IF

(* Outputs *)
ACT_Output_To_Device_And_User;
ACT_Build_StatusMessage;

END_FUNCTION_BLOCK

ACTIONS
	ACTION ACT_Init

		IF StateEntry THEN
	    (* Timeout starten *)
	   		t_init_timeout(IN := TRUE, PT := init_timeout);
	    END_IF

	    (* Seriennummer vom Gerät lesen *)
	    Output_DeviceInstance.serialnumber := Input_SN;

	    (* Plausibilitätsprüfung *)
	    sn_valid := (LEN(Input_SN) >= 4) AND (Input_SN <> '0000');

	    IF sn_valid THEN
	        (* Verbindung erfolgreich *)
	        t_init_timeout(IN := FALSE);
	        Output_DeviceInstance.status_msg := CONCAT('Device connection established. SN=', Input_SN);

			(* Erstmaligen Status abrufen *)
		    cfg_pending := TRUE;

		    ACT_device_type_feedback;
		    ACT_cfg_mode_feedback;

		    Output_ErrorState := DEV_ERR_NONE;
		    state_next := DV_IDLE;
	    END_IF

	    (* Timeout abgelaufen -> Fehler *)
	    IF t_init_timeout.Q THEN
			Output_ErrorState := DEV_ERR_INIT;
	        Output_DeviceInstance.status_msg := 'ERROR: Device connection timeout – no valid serial number';
	        state_next := DV_ERROR;
	    END_IF

	END_ACTION

	ACTION ACT_Latch_Reset

		(* ERROR Reset *)

		req_reset := Input_DeviceInstance.reset;
		Input_DeviceInstance.reset := FALSE;
		Output_DeviceInstance.reset := FALSE;
	END_ACTION

	ACTION ACT_Latch_ControlMode
	    (* ControlMode *)
	    IF Input_DeviceInstance.control_mode_req <> Input_ControlMode THEN
	        cfg_mode_req := Input_DeviceInstance.control_mode_req;
	        cfg_pending := TRUE;
	    END_IF
	    cfg_mode_act := Input_ControlMode;

	    setpoint_mode_allowed := (cfg_mode_act = 0);   (* 0 = BUS/RS232 *)

	    IF NOT setpoint_mode_allowed THEN
	    	ACT_Central_SVreq_Discard;
	    END_IF
	END_ACTION

	ACTION ACT_Latch_SVreq
	    (* SV Requests *)
	    IF NOT cfg_pending AND setpoint_mode_allowed THEN

	    	CASE Input_DeviceType OF

	    	ELFLOW, CORIFLOW:
	    		sv_changed := ABS(Input_DeviceInstance.SVreq - Input.SV) >= 0.001;
	    	ELPRESS:
				sv_changed := ABS(Input_DeviceInstance.SVreq - Input_p_SV_mbarg) >= 1.0;

	    	END_CASE

			IF sv_changed THEN
	            sv_req := Input_DeviceInstance.SVreq;
	            ACT_Reset_SV_Lifecycle;	(* Lebenszyklus neu starten *)
	            sv_pending := TRUE;
	        END_IF

	    END_IF

	END_ACTION

	ACTION ACT_Reset_SV_Lifecycle
		sv_rejected := FALSE;
	    sv_applied  := FALSE;
	    sv_accepted := FALSE;
	    sv_reached  := FALSE;
	    sv_maintained := FALSE;

	    t_sv_accept(IN := FALSE);
		t_av_timeout(IN := FALSE);
		t_av_NOTmaintained(IN := FALSE);

	END_ACTION

	ACTION ACT_Controlling
			(* === CONTROLLING: Überwachung === *)

	        (* Timeout *)
	        t_av_timeout(IN := NOT sv_reached, PT := Input_AV_Timeout);

	        IF t_av_timeout.Q THEN
	        	RETURN;
	        END_IF

	        (* Toleranzprüfung *)
	        AV_lower_range_limit := activePrimary.SVreq * (100.0-(SV_tolerance*0.5))/100.0;
			AV_upper_range_limit := activePrimary.SVreq * (100.0+(SV_tolerance*0.5))/100.0;

			AV_in_range := INRANGE(AV_lower_range_limit,activePrimary.AV,AV_upper_range_limit);

	        IF AV_in_range THEN
	            sv_reached := TRUE;
	        ELSE
	        	sv_reached := FALSE;
	        END_IF

	END_ACTION

	ACTION ACT_Settled
			(* Timeout *)
	    	t_av_NOTmaintained(IN := NOT sv_maintained, PT := T#10s); (* Variabel über User !!*)

	        (* Rückfall, falls Wert wieder wegdriftet *)
	        AV_lower_range_limit := activePrimary.SVreq * (100.0-(SV_tolerance*1))/100.0;
			AV_upper_range_limit := activePrimary.SVreq * (100.0+(SV_tolerance*1))/100.0;

			AV_in_range := INRANGE(AV_lower_range_limit,activePrimary.AV,AV_upper_range_limit);
	        IF AV_in_range THEN
	        	sv_maintained := TRUE;
	        ELSE
	        	sv_maintained := FALSE;
	        END_IF
	END_ACTION

	ACTION ACT_Central_SVreq_Discard

        sv_pending := FALSE;

        (* SV-Latches zurücksetzen *)
		sv_req := 0.0;

        (* Lebenszyklus vollständig zurücksetzen *)
        ACT_Reset_SV_Lifecycle;

        (* Rückmeldung an User *)
        Output_DeviceInstance.SVreq := 0.0;

		(* Device Reset zurücksetzten *)
		Output_Reset_to_device := 0;
	END_ACTION

	ACTION ACT_device_type_feedback
			CASE Input_DeviceType OF
				ELFLOW:   dv_str := ': ELFLOW';
				CORIFLOW: dv_str := ': CoriFlow';
				ELPRESS:  dv_str := ': ELPRESS';
			ELSE
				dv_str := ' - undefined';
			END_CASE
	END_ACTION

	ACTION ACT_pInput_bara_to_mbarg
		Input_p_SV_mbarg := Input.SV*1000-1000; (* mbar(g) *)
		Input_p_AV_mbarg := Input.AV*1000-1000; (* mbar(a) *)
	END_ACTION

	ACTION ACT_cfg_mode_feedback
		CASE cfg_mode_act OF
			0: cm_str := 'BUS/RS232';
			1: cm_str := 'Analog input';
			2: cm_str := 'FLOW-BUS slave';
			3: cm_str := 'Valve close';
			4: cm_str := 'Controller idle';
			5: cm_str := 'Testing mode';
			6: cm_str := 'Tuning mode';
			7: cm_str := 'Setpoint 100%';
			8: cm_str := 'Valve fully open';
			9: cm_str := 'Calibration mode';
			10: cm_str := 'Analog slave';
			12: cm_str := 'setpoint 0%';
			13: cm_str := 'FLOW-BUS analog slave';
			18: cm_str := 'RS232';
			20: cm_str := 'valve steering (valve = setpoint)';
			21: cm_str := 'analog valve steering(valve = analog input)';
			22: cm_str := 'valve safe state';
		ELSE
            cm_str := ' - undefined';
		END_CASE
	END_ACTION

	ACTION ACT_SelectActiveChannel
		activePrimary.SVreq := sv_req;
		activePrimary.AV := Input.AV;
		activePrimary.DeviceSV := Input.SV;
		activePrimary.Unit := Input.Unit;
		activePrimary.SV_Min := Input_DeviceInstance.lower_limit;
		activePrimary.SV_Max := Input_DeviceInstance.upper_limit;

		CASE Input_DeviceType OF

		ELFLOW,CORIFLOW: (* Flow *)
			activePrimary.SVreq := sv_req;
			activePrimary.AV := Input.AV;
			activePrimary.DeviceSV := Input.SV;
			activePrimary.Unit := Input.Unit;
			activePrimary.SV_Min := Input_DeviceInstance.lower_limit;
			activePrimary.SV_Max := Input_DeviceInstance.upper_limit;
		ELPRESS: (* Pressure *)
			activePrimary.SVreq := sv_req;
			activePrimary.AV := Input_p_AV_mbarg;
			activePrimary.DeviceSV := Input_p_SV_mbarg;
			activePrimary.Unit := Input_p_unit_mbarg;
			activePrimary.SV_Min := 0.0;
			activePrimary.SV_Max := P_MAX_BAR;

		END_CASE

		sv_active := (activePrimary.SVreq <> 0.0);
	END_ACTION

	ACTION ACT_Commit_Config

	    IF cfg_pending THEN

			 (* === Commit ControlMode === *)
	        Output_ControlMode := cfg_mode_req;

			IF Input_ControlMode = cfg_mode_req THEN
		        ACT_cfg_mode_feedback;
		        cfg_pending := FALSE;
	        END_IF

	    END_IF

	END_ACTION

	ACTION ACT_Handle_SV

		IF NOT setpoint_mode_allowed THEN
		    sv_rejected := TRUE;
		    sv_rejected_latched := TRUE;
		    RETURN;
		END_IF

	    (* Nur relevante States *)
	    IF (state <> DV_SETTING_REQ) AND
	       (state <> DV_CONTROLLING) AND
	       (state <> DV_SETTLED) THEN
	        sv_rejected := TRUE;
	        sv_rejected_latched := TRUE;
	        RETURN;
	    END_IF

	    (* Keine Arbeit bei Config-Wechsel *)
	    IF cfg_pending THEN
	    	sv_rejected := TRUE;
	    	sv_rejected_latched := TRUE;
	        RETURN;
	    END_IF

		sv_str := CONCAT(REAL_TO_STRING(activePrimary.SVreq), activePrimary.Unit);

		IF NOT sv_applied THEN

	        (* Bereich prüfen *)
			SV_in_range := INRANGE(activePrimary.SV_Min, activePrimary.SVreq, activePrimary.SV_Max);

			IF NOT SV_in_range THEN
			    (* === Ungültigen User-Sollwert zurückweisen === *)

			    sv_pending := FALSE;

				IF activePrimary.SVreq < activePrimary.SV_Min OR activePrimary.SVreq > activePrimary.SV_Max THEN
				    (* User-SV auf aktuell gültigen Sollwert zurücksetzen *)
				    ACT_Restore_UserSetpoints;

				    (* Optional: Statusmeldung *)
				    sv_outofrange := TRUE;
					sv_rejected := TRUE;
					sv_rejected_latched := TRUE;

				    RETURN;
				  END_IF
			END_IF

			sv_outofrange := FALSE;
			sv_rejected_latched := FALSE;
	        sv_applied := TRUE;
	        sv_pending := FALSE;
		END_IF

		(* Prüfen, ob Gerät SV übernommen hat *)
		IF sv_applied AND NOT sv_accepted THEN
			(* Akzeptanz-Timer starten *)
		    t_sv_accept(IN := TRUE, PT := Input_SV_Accept_Timeout);

			IF ABS(activePrimary.SVreq - activePrimary.DeviceSV) <= activePrimary.SVreq * 0.01 THEN
				sv_accepted := TRUE;
			END_IF

		END_IF

	END_ACTION

	ACTION ACT_Restore_UserSetpoints
		 Output_DeviceInstance.SVreq := sv_req;
	END_ACTION

	ACTION ACT_Output_To_Device_And_User

	    (* ================================================= *)
	    (* Default: keine Sollwerte an das Gerät             *)
	    (* ================================================= *)
	    CASE Input_DeviceType OF

		ELFLOW,CORIFLOW: (* Flow *)
			    Output_SVreq := 0.0;
	    ELPRESS: (* Pressure *)
	    		Output_SVreq := 1.0;

		END_CASE

	    (* ================================================= *)
	    (* Sollwert nur ausgeben, wenn er gültig angewandt    *)
	    (* ================================================= *)
	    IF sv_applied AND
	       (state = DV_SETTING_REQ OR state = DV_CONTROLLING OR state = DV_SETTLED) THEN

	       CASE Input_DeviceType OF

	            ELFLOW,CORIFLOW:  (* Flow *)
	            	Output_SVreq := sv_req;

	            ELPRESS: (* Pressure *)
	                Output_SVreq := sv_req/1000+1; (* Umrechnung von mbar (g) zu bar (a) *)

	        END_CASE

	    END_IF

	    (* ================================================= *)
	    (* Status an User                                    *)
	    (* ================================================= *)
		ACT_ReadAV;

	    Output_DeviceInstance.control_mode     := cfg_mode_act;
	    Output_DeviceInstance.control_mode_req     := cfg_mode_req;

		Output_DeviceInstance.state := state;
		Output_DeviceInstance.enable := Input_DeviceInstance.enable;
		Output_DeviceInstance.SVaccepted := sv_accepted;
		Output_DeviceInstance.SVrejected := sv_rejected;
		Output_DeviceInstance.SVreached := sv_reached;
		CASE Input_DeviceType OF

		ELFLOW,CORIFLOW: (* Flow *)
			    Output_DeviceInstance.SVreq := sv_req;
			    Output_DeviceInstance.SV := Input.SV;
	    ELPRESS: (* Pressure *)
	    		Output_DeviceInstance.SVreq := sv_req;
				Output_DeviceInstance.SV := Input_p_SV_mbarg;

		END_CASE

	END_ACTION

	ACTION ACT_Map_AlarmInfo
	    Output_DeviceInstance.alarm_info := Input_alarm_info;
	END_ACTION

	ACTION ACT_ReadAV
		Output_DeviceInstance.media := Input_FluidName;

(*		CASE Input_DeviceType OF *)
(*		 *)
(*		CORIFLOW, ELFLOW: *)
(*				IF Input.AV > Input_DeviceInstance.upper_limit / 500.0 THEN *)
(*					Output_DeviceInstance.AV := Input.AV; *)
(*				ELSE *)
(*					Output_DeviceInstance.AV := 0.0; *)
(*				END_IF; *)
(*		ELPRESS: *)
(*				IF Input_p_AV_mbarg > Input_DeviceInstance.upper_limit / 500.0 THEN *)
(*				    Output_DeviceInstance.AV := Input_p_AV_mbarg; *)
(*				ELSE *)
(*				    Output_DeviceInstance.AV := 0.0; *)
(*				END_IF; *)
(*		END_CASE *)

		Output_DeviceInstance.AV := activePrimary.AV;

		Output_DeviceInstance.unit := Input.Unit;
		Output_DeviceInstance.serialnumber := Input_SN;
		Output_DeviceInstance.name := Input_UserTag;

		Output_DeviceInstance.temperature := Input_temperature;
		Output_DeviceInstance.density := Input_density;
	END_ACTION

	ACTION ACT_ProcessAlarmInfo_Input
		Input_alarm_info := BH_AlarmBitTOAlarmArray(Input.AlarmInfo);
	END_ACTION

	ACTION ACT_AlarmInfo_wo_text

	    FLAG_Alarm := FALSE;
	    FLAG_Warning := FALSE;

		warning_detail_str := '';

	    FOR k := 1 TO 8 DO
	        IF Output_DeviceInstance.alarm_info[k] THEN

	            CASE k OF
	                1: (* Alarm *)
	                    FLAG_Alarm := TRUE;

	                2: (* Warning *)
	                    FLAG_Warning := TRUE;

	                3: (* Sensor < min *)
	                    FLAG_Warning := TRUE;
	                    warning_detail_str := CONCAT(warning_detail_str, 'Sensor below minimum limit; ');

	                4: (* Sensor > max *)
	                    FLAG_Warning := TRUE;
	                    warning_detail_str := CONCAT(warning_detail_str, 'Sensor above maximum limit; ');

	                5: (* Batch counter *)
	                    FLAG_Warning := TRUE;
	                    warning_detail_str := CONCAT(warning_detail_str, 'Batch counter limit reached; ');

	                6: (* Power-up / deviation *)
	                    FLAG_Warning := TRUE;
	                    warning_detail_str := CONCAT(warning_detail_str, 'Power-up alarm; ');

	                7: (* Communication *)
	                    FLAG_Alarm := TRUE;
	                    Output_ErrorState := DEV_ERR_COMMUNICATION;
	                8: (* Hardware *)
	                    FLAG_Alarm := TRUE;
	                    Output_ErrorState := DEV_ERR_HARDWARE;

	            END_CASE
	        END_IF
	    END_FOR

	    Output_DeviceInstance.warning := FLAG_Warning;
	    Output_DeviceInstance.alarm   := FLAG_Alarm;

	END_ACTION

	ACTION ACT_Status_wo_text

        Output_DeviceInstance.status := Input_status;

        (* Default zurücksetzen *)
        (* Wichtig: nicht alarm/warning global löschen! *)

        CASE Input_status OF

            0: (* Normal operation *)
                ;(* nichts setzen *)

            1: (* Maintenance required *)
                Output_DeviceInstance.warning := TRUE;

            2: (* Out of specification *)
                Output_DeviceInstance.warning := TRUE;

            4: (* Check function *)
                Output_DeviceInstance.warning := TRUE;

            8: (* Device failure *)
                Output_DeviceInstance.alarm := TRUE;
                FLAG_Alarm := TRUE;
                Output_ErrorState := DEV_ERR_DEVICE_FAILURE;

            ELSE
                (* unbekannter Status *)
                Output_DeviceInstance.warning := TRUE;

        END_CASE

	END_ACTION

	ACTION ACT_Name

		IF Input_UserTag <> Output_DeviceInstance.name THEN
			Output_UserTag := Output_DeviceInstance.name;
			Output_DeviceInstance.name := Output_DeviceInstance.name;
		END_IF

	END_ACTION

	ACTION ACT_Build_StatusMessage

	    Output_DeviceInstance.status_msg := '';

	    (* === Priority Prefix === *)
	    IF state = DV_INIT THEN
	        Output_DeviceInstance.status_msg :=
	            CONCAT(notification_lable, 'Initializing device...');
	        RETURN;
	    END_IF

    	CASE Output_ErrorState OF

    		DEV_ERR_NONE: err_msg := '';

    		DEV_ERR_INIT: err_msg := 'Initialization timeout';

    		DEV_ERR_SV_ACCEPT_TIMEOUT: err_msg := 'Set Value not accepted - TIMEOUT';

    		DEV_ERR_AV_Reach_TIMEOUT: err_msg := 'Actual Value not in tolerance - TIMEOUT';

    		DEV_ERR_AV_Maintain_TIMEOUT: err_msg := 'Actual Value not maintained - TIMEOUT';

    		DEV_ERR_COMMUNICATION: err_msg := 'Communication error';

    		DEV_ERR_HARDWARE: err_msg := 'Hardware alarm';

    		DEV_ERR_DEVICE_FAILURE: err_msg := 'Device failure';

    	END_CASE

		IF sv_rejected_latched THEN
			Output_DeviceInstance.warning := TRUE;
			IF warning_detail_str <> '' THEN
				warning_detail_str := CONCAT(warning_detail_str, ', Setpoint rejected - ');
			ELSE
				warning_detail_str := 'Setpoint rejected - ';
			END_IF

			IF NOT setpoint_mode_allowed THEN
				warning_detail_str := CONCAT(warning_detail_str, 'no Setpoint allowed.');
			ELSIF cfg_pending THEN
				warning_detail_str := CONCAT(warning_detail_str, 'HW-Config pending.');
			ELSIF sv_outofrange THEN
				warning_detail_str := CONCAT(warning_detail_str, 'Setpoint out of range.');
			END_IF

		END_IF

	    IF Output_DeviceInstance.alarm THEN
	        prefix := alarm_lable;
	    ELSIF state = DV_ERROR THEN
	    	prefix := error_lable;
	    ELSIF Output_DeviceInstance.warning THEN
	        prefix := warning_lable;
	    ELSE
	        prefix := notification_lable;
	    END_IF

	    Output_DeviceInstance.status_msg := prefix;

	    (* === ControlFunction / ControlMode === *)
	    Output_DeviceInstance.status_msg :=
	        CONCAT(Output_DeviceInstance.status_msg, 'DV=');
	    Output_DeviceInstance.status_msg :=
	        CONCAT(Output_DeviceInstance.status_msg, dv_str);

		Output_DeviceInstance.status_msg :=
	        CONCAT(Output_DeviceInstance.status_msg, ', CM=');
	    Output_DeviceInstance.status_msg :=
	        CONCAT(Output_DeviceInstance.status_msg, cm_str);

	    (* === Setpoint === *)
	    IF sv_applied THEN
	        Output_DeviceInstance.status_msg :=
		        CONCAT(Output_DeviceInstance.status_msg, ', SV=');
		    Output_DeviceInstance.status_msg :=
		        CONCAT(Output_DeviceInstance.status_msg, sv_str);
	    END_IF

	    (* === State-dependent text === *)
	    CASE state OF
	        DV_IDLE:
	            msg_str := ' (Idle)';
	        DV_SETTING_REQ:
	            IF sv_accepted THEN
	                msg_str := ' (Setpoint accepted)';
	            ELSE
	                msg_str := ' (Waiting for device to accept setpoint)';
	            END_IF
	        DV_CONTROLLING:
	            msg_str := ' (Controlling)';
	        DV_SETTLED:
	            msg_str := ' (Setpoint reached)';
	        DV_DISABLED:
	            msg_str := ' (Disabled)';
	    ELSE
	        msg_str := '';
	    END_CASE

	    CASE Output_DeviceInstance.status OF
		    0:
		        dev_status_str := 'Normal operation';

		    1:
		        dev_status_str := 'Maintenance required';

		    2:
		        dev_status_str := 'Out of specification';

		    4:
		        dev_status_str := 'Check function';

		    8:
		        dev_status_str := 'Device failure';

		ELSE
		    dev_status_str := 'Unknown device status';
		END_CASE

	    Output_DeviceInstance.status_msg :=
	        CONCAT(Output_DeviceInstance.status_msg, msg_str);

		Output_DeviceInstance.status_msg :=
	        CONCAT(Output_DeviceInstance.status_msg, ' | Status: ');
	    Output_DeviceInstance.status_msg :=
	        CONCAT(Output_DeviceInstance.status_msg, dev_status_str);

		IF err_msg <> '' THEN
    		Output_DeviceInstance.status_msg := CONCAT(Output_DeviceInstance.status_msg, ' | ');
    		Output_DeviceInstance.status_msg := CONCAT(Output_DeviceInstance.status_msg, error_lable);
        	Output_DeviceInstance.status_msg := CONCAT(Output_DeviceInstance.status_msg, err_msg);
	    END_IF

	    IF warning_detail_str <> '' THEN
	    	Output_DeviceInstance.status_msg := CONCAT(Output_DeviceInstance.status_msg, ' | ');
	    	Output_DeviceInstance.status_msg := CONCAT(Output_DeviceInstance.status_msg, warning_detail_str);
	    END_IF
	END_ACTION

	ACTION ACT_Reset_BH_Device
		Output_Reset_Alarm_Enable := Input_DeviceInstance.alarm_reset_enable;
		IF Input_AlarmMode = 4 THEN
			Output_Reset_to_device := 2; (* reset alarm *)
			msg_str := ': Device reset triggered.';
		    Output_DeviceInstance.status_msg := CONCAT(notification_lable, Input_DeviceInstance.name);
		    Output_DeviceInstance.status_msg := CONCAT(Output_DeviceInstance.status_msg, msg_str);
		    Output_DeviceInstance.reset := FALSE;
		 ELSE
		 	msg_str := ': Device reset NOT available.';
		    Output_DeviceInstance.status_msg := CONCAT(warning_lable, Input_DeviceInstance.name);
		    Output_DeviceInstance.status_msg := CONCAT(Output_DeviceInstance.status_msg, msg_str);
		 END_IF

	END_ACTION

END_ACTIONS

(* ---- FB_CAN_Broker.st ---- *)
 (********************************************************************************
 * FUNCTION_BLOCK: FB_CAN_Broker
 *
 * Beschreibung:
 *   Zentraler Hardware-Treiber-Manager für den CAN-Bus an Bachmann M1 (CUL_PLC).
 *
 *   Aufgaben:
 *     1. Kapselt den Hardware-Zugriff (CardNb, NetNb, Chan, CUL_PLC).
 *     2. Liest in jedem SPS-Zyklus die Hardware-Empfangsqueue vollständig leer
 *        und verteilt empfangene Telegramme an den passenden Kanal.
 *     3. Verwaltet Sendeaufträge über ein faires Round-Robin-Verfahren
 *        (nicht-blockierend über CUL_SendMsg_NB), sodass keine Buskollisionen entstehen.
 ********************************************************************************)
FUNCTION_BLOCK FB_CAN_Broker
VAR_INPUT
    Enable          : BOOL := TRUE;             (* Broker aktivieren *)
    Reset           : BOOL := FALSE;            (* Re-Init auslösen *)
    NetNb           : DINT := 1;                (* CAN NetNumber (Standard: 1) *)
    CardNb          : DINT := 2;                (* CPU Card Number (Card 2) *)
    Chan            : UDINT := 0;               (* CAN-Kanal (0 = CAN A) *)
END_VAR

VAR_IN_OUT
    Channel1        : ST_CAN_Broker_Channel;    (* Kanal für Sensor 1 *)
    Channel2        : ST_CAN_Broker_Channel;    (* Kanal für Sensor 2 *)
    Channel3        : ST_CAN_Broker_Channel;    (* Kanal für Sensor 3 *)
END_VAR

VAR_OUTPUT
    Ready           : BOOL := FALSE;            (* Treiber initialisiert und empfangsbereit *)
    Error           : BOOL := FALSE;            (* Treiberfehler *)
    ErrorID         : DINT := 0;
END_VAR

VAR
    initStep        : INT := 0;
    initDone        : BOOL := FALSE;

    (* CUL Instanzen *)
    fbAttachEvent   : CUL_AttachEvent;
    fbSendMsg       : CUL_SendMsg_NB;
    fbRecvMsg       : CUL_ReceiveMsg;

    dwEventFlags    : UDINT := 0;
    nRet            : DINT := 0;

    (* Dynamische Rx-ID-Registrierung *)
    lastEnabledRx1  : UDINT := 0;
    lastEnabledRx2  : UDINT := 0;
    lastEnabledRx3  : UDINT := 0;

    (* Sende-Verwaltung *)
    txActive        : BOOL := FALSE;
    activeChan      : INT := 0;                 (* 1, 2 oder 3 *)
    lastServedChan  : INT := 1;
    currTxCobId     : UDINT := 0;
    currTxData      : ARRAY [0..7] OF BYTE;

    (* Hilfsvariablen *)
    i               : INT;
    candChan        : INT;
    rxCount         : INT;
END_VAR

(* ============================================================================ *)
(* Deaktivierung & Reset                                                       *)
(* ============================================================================ *)
IF NOT Enable THEN
    IF initDone THEN
        Cul_DetachEvent(NetNb := NetNb, Event := 0);
    END_IF;
    Ready    := FALSE;
    initDone := FALSE;
    initStep := 0;
    txActive := FALSE;
    RETURN;
END_IF;

IF Reset THEN
    IF initDone THEN
        Cul_DetachEvent(NetNb := NetNb, Event := 0);
    END_IF;
    Ready          := FALSE;
    Error          := FALSE;
    ErrorID        := 0;
    initDone       := FALSE;
    initStep       := 0;
    txActive       := FALSE;
    lastEnabledRx1 := 0;
    lastEnabledRx2 := 0;
    lastEnabledRx3 := 0;
END_IF;

(* ============================================================================ *)
(* Initialisierung der Hardware (Schritt 0)                                     *)
(* ============================================================================ *)
IF NOT initDone THEN
    CASE initStep OF
        0:
            (* Alle 3 Antwort-IDs freischalten *)
            IF Channel1.RxCobId > 0 AND Channel1.RxCobId <> lastEnabledRx1 THEN
                nRet := Cul_EnableMsg(CardNb := CardNb, Chan := Chan, CobId := Channel1.RxCobId);
                lastEnabledRx1 := Channel1.RxCobId;
            END_IF;
            IF Channel2.RxCobId > 0 AND Channel2.RxCobId <> lastEnabledRx2 THEN
                nRet := Cul_EnableMsg(CardNb := CardNb, Chan := Chan, CobId := Channel2.RxCobId);
                lastEnabledRx2 := Channel2.RxCobId;
            END_IF;
            IF Channel3.RxCobId > 0 AND Channel3.RxCobId <> lastEnabledRx3 THEN
                nRet := Cul_EnableMsg(CardNb := CardNb, Chan := Chan, CobId := Channel3.RxCobId);
                lastEnabledRx3 := Channel3.RxCobId;
            END_IF;

            dwEventFlags := 0;
            fbAttachEvent(Req := TRUE, NetNb := NetNb, Event := dwEventFlags);

            IF fbAttachEvent.Done THEN
                fbAttachEvent(Req := FALSE, NetNb := NetNb, Event := dwEventFlags);
                initDone := TRUE;
                Ready    := TRUE;
                Error    := FALSE;
                ErrorID  := 0;
            ELSIF fbAttachEvent.Error THEN
                Error    := TRUE;
                ErrorID  := fbAttachEvent.Status;
            END_IF;
    END_CASE;
    RETURN;
END_IF;

(* Nachträglich konfigurierte oder geänderte RxCobIds beim CAN-Controller freischalten *)
IF Channel1.RxCobId > 0 AND Channel1.RxCobId <> lastEnabledRx1 THEN
    nRet := Cul_EnableMsg(CardNb := CardNb, Chan := Chan, CobId := Channel1.RxCobId);
    lastEnabledRx1 := Channel1.RxCobId;
END_IF;
IF Channel2.RxCobId > 0 AND Channel2.RxCobId <> lastEnabledRx2 THEN
    nRet := Cul_EnableMsg(CardNb := CardNb, Chan := Chan, CobId := Channel2.RxCobId);
    lastEnabledRx2 := Channel2.RxCobId;
END_IF;
IF Channel3.RxCobId > 0 AND Channel3.RxCobId <> lastEnabledRx3 THEN
    nRet := Cul_EnableMsg(CardNb := CardNb, Chan := Chan, CobId := Channel3.RxCobId);
    lastEnabledRx3 := Channel3.RxCobId;
END_IF;

(* ============================================================================ *)
(* Zyklus-Start: Flanken / Trigger der Kanäle zurücksetzen                      *)
(* ============================================================================ *)
Channel1.RxNew  := FALSE;
Channel1.TxDone := FALSE;
Channel1.TxError:= FALSE;

Channel2.RxNew  := FALSE;
Channel2.TxDone := FALSE;
Channel2.TxError:= FALSE;

Channel3.RxNew  := FALSE;
Channel3.TxDone := FALSE;
Channel3.TxError:= FALSE;

(* ============================================================================ *)
(* 1. EMPFANG: Hardware-Queue vollständig auslesen & an Kanäle verteilen        *)
(* ============================================================================ *)
rxCount := 0;
REPEAT
    fbRecvMsg(NetNb := NetNb);
    rxCount := rxCount + 1;

    IF fbRecvMsg.Status = 0 AND fbRecvMsg.Msg_Length >= 7 THEN
        IF fbRecvMsg.CobId = Channel1.RxCobId THEN
            Channel1.RxNew  := TRUE;
            Channel1.RxData := fbRecvMsg.Msg_Data;
            Channel1.RxLen  := fbRecvMsg.Msg_Length;
        ELSIF fbRecvMsg.CobId = Channel2.RxCobId THEN
            Channel2.RxNew  := TRUE;
            Channel2.RxData := fbRecvMsg.Msg_Data;
            Channel2.RxLen  := fbRecvMsg.Msg_Length;
        ELSIF fbRecvMsg.CobId = Channel3.RxCobId THEN
            Channel3.RxNew  := TRUE;
            Channel3.RxData := fbRecvMsg.Msg_Data;
            Channel3.RxLen  := fbRecvMsg.Msg_Length;
        END_IF;
    END_IF;
UNTIL (fbRecvMsg.Status <> 0) OR (fbRecvMsg.Msg_Left = 0) OR (rxCount > 15)
END_REPEAT;

(* ============================================================================ *)
(* 2. SENDEN: Laufende Übertragung überwachen oder neuen Auftrag starten        *)
(* ============================================================================ *)
IF txActive THEN
    (* Laufenden Sendevorgang pollen *)
    fbSendMsg(
        Req        := TRUE,
        NetNb      := NetNb,
        CobId      := currTxCobId,
        Msg_Data   := currTxData,
        Msg_Length := 8
    );

    IF fbSendMsg.Done THEN
        fbSendMsg(Req := FALSE, NetNb := NetNb, CobId := currTxCobId, Msg_Data := currTxData, Msg_Length := 8);
        txActive := FALSE;
        CASE activeChan OF
            1: Channel1.TxDone := TRUE; Channel1.TxBusy := FALSE; Channel1.TxReq := FALSE;
            2: Channel2.TxDone := TRUE; Channel2.TxBusy := FALSE; Channel2.TxReq := FALSE;
            3: Channel3.TxDone := TRUE; Channel3.TxBusy := FALSE; Channel3.TxReq := FALSE;
        END_CASE;
    ELSIF fbSendMsg.Error THEN
        fbSendMsg(Req := FALSE, NetNb := NetNb, CobId := currTxCobId, Msg_Data := currTxData, Msg_Length := 8);
        txActive := FALSE;
        CASE activeChan OF
            1: Channel1.TxError := TRUE; Channel1.TxBusy := FALSE; Channel1.TxReq := FALSE;
            2: Channel2.TxError := TRUE; Channel2.TxBusy := FALSE; Channel2.TxReq := FALSE;
            3: Channel3.TxError := TRUE; Channel3.TxBusy := FALSE; Channel3.TxReq := FALSE;
        END_CASE;
    END_IF;

ELSE
    (* Kein Sendevorgang aktiv: Nächsten Sendeauftrag per Round-Robin auswählen *)
    FOR i := 1 TO 3 DO
        candChan := ((lastServedChan - 1 + i) MOD 3) + 1;

        IF candChan = 1 AND Channel1.TxReq THEN
            activeChan      := 1;
            lastServedChan  := 1;
            currTxCobId     := Channel1.TxCobId;
            currTxData      := Channel1.TxData;
            Channel1.TxBusy := TRUE;
            txActive        := TRUE;
            EXIT;
        ELSIF candChan = 2 AND Channel2.TxReq THEN
            activeChan      := 2;
            lastServedChan  := 2;
            currTxCobId     := Channel2.TxCobId;
            currTxData      := Channel2.TxData;
            Channel2.TxBusy := TRUE;
            txActive        := TRUE;
            EXIT;
        ELSIF candChan = 3 AND Channel3.TxReq THEN
            activeChan      := 3;
            lastServedChan  := 3;
            currTxCobId     := Channel3.TxCobId;
            currTxData      := Channel3.TxData;
            Channel3.TxBusy := TRUE;
            txActive        := TRUE;
            EXIT;
        END_IF;
    END_FOR;

    IF txActive THEN
        fbSendMsg(
            Req        := TRUE,
            NetNb      := NetNb,
            CobId      := currTxCobId,
            Msg_Data   := currTxData,
            Msg_Length := 8
        );
    END_IF;
END_IF;

END_FUNCTION_BLOCK

(* ---- FB_microFlow_Device.st ---- *)
(********************************************************************************
 * FUNCTION_BLOCK: FB_microFlow_Device
 *
 * Beschreibung:
 *   Modularer, gerätespezifischer Treiberbaustein für einen einzelnen
 *   microFlow Gas-Sensor (Wi.Tec).
 *
 *   Highlights:
 *     1. Auto-Discovery beim Initialisieren:
 *        Liest Seriennummer, Firmware, Gastyp (z.B. CO, CO2), Messbereich (z.B. 50.0)
 *        und Einheit (ppm / Vol.%) vollautomatisch aus dem Sensor aus!
 *     2. Volle Zustandsmaschine (State Machine) nach Industriestandard.
 *     3. Automatische Übernahme und Klartext-Meldung von Gerätefehlern
 *        (z.B. IR-Signalpegel < 50%, Strahler fehlt, UV-Pegelfehler, Timeout).
 *     4. Trennung von Treiber und Logik: Kommuniziert über ST_CAN_Broker_Channel.
 ********************************************************************************)
FUNCTION_BLOCK FB_microFlow_Device
VAR_INPUT
    Enable              : BOOL := TRUE;         (* Sensor-Baustein aktivieren *)
    Reset               : BOOL := FALSE;        (* Fehler-Quittierung / Re-Init *)

    (* Adressierung *)
    Tx_CobId            : UDINT := 16#300;      (* Sende-ID an diesen Sensor *)
    Rx_CobId            : UDINT := 16#208;      (* Empfangs-ID von diesem Sensor *)

    (* Abtastraten *)
    PollInterval_Conc   : TIME := T#100ms;      (* Schnelle Abtastung Konzentration (z.B. 100ms = 10Hz) *)
    PollInterval_Temp   : TIME := T#5s;         (* Langsame Abtastung Temperatur (alle 5 Sekunden) *)
    TimeoutTime         : TIME := T#150ms;      (* Wartezeit auf Antwort *)
    ReadCH2             : BOOL := FALSE;        (* Kanal 2 ebenfalls abfragen *)

    (* Steuerbefehle *)
    Cmd_ZeroCalibration : BOOL := FALSE;        (* Flanke startet Nullpunkt-Kalibrierung (Cmd 16#11) *)
    Cmd_ResetDevice     : BOOL := FALSE;        (* Flanke startet Software-Reset des Sensors (Cmd 16#04) *)
END_VAR

VAR_IN_OUT
    Bus                 : ST_CAN_Broker_Channel; (* Verbindung zum zentralen CAN-Broker *)
END_VAR

VAR_OUTPUT
    Data                : ST_microFlow_Data;    (* Sämtliche Messwerte, Gerätedaten und Fehler *)
END_VAR

VAR
    (* Zustandssteuerung *)
    eState              : E_microFlow_State := MF_STATE_DISABLED;
    subStep             : INT := 0;             (* 0=Send, 1=Wait *)
    queryCH2Active      : BOOL := FALSE;
    timeoutCounter      : INT := 0;

    (* Flankenerkennung für Befehle *)
    oldZeroCalib        : BOOL := FALSE;
    oldResetDev         : BOOL := FALSE;

    (* Timer *)
    tPollConc           : TON;
    tPollTemp           : TON;
    tTimeout            : TON;

    (* Helfer für Float & Integer *)
    dwHelper            : DWORD;
    pRealHelper         : POINTER TO REAL;
    nUnitVal            : UINT;
    nGasIdx             : USINT;
END_VAR

(* ============================================================================ *)
(* Bus-Kanal-IDs synchronisieren                                               *)
(* ============================================================================ *)
Bus.TxCobId := Tx_CobId;
Bus.RxCobId := Rx_CobId;

(* ============================================================================ *)
(* Baustein-Deaktivierung                                                      *)
(* ============================================================================ *)
IF NOT Enable THEN
    eState          := MF_STATE_DISABLED;
    Data.State      := MF_STATE_DISABLED;
    Data.StateText  := 'Deaktiviert';
    Data.Connected  := FALSE;
    Bus.TxReq       := FALSE;
    subStep         := 0;
    RETURN;
END_IF;

(* ============================================================================ *)
(* Fehler-Reset                                                                *)
(* ============================================================================ *)
IF Reset THEN
    Data.Error      := FALSE;
    Data.ErrorCode  := MF_ERR_NONE;
    Data.ErrorText  := 'OK';
    timeoutCounter  := 0;
    subStep         := 0;
    eState          := MF_STATE_INIT_START;
END_IF;

(* ============================================================================ *)
(* Kontinuierliche Übernahme von Gerätefehlern aus dem Statusbyte              *)
(* ============================================================================ *)
IF Bus.RxNew AND Bus.RxLen >= 7 THEN
    Data.StatusByte      := Bus.RxData[6];

    (* Bit-Zuordnung laut microFlow Handbuch S. 9 *)
    Data.IR_Detected     := (Data.StatusByte AND 16#80) <> 16#00; (* Bit 7: 1 = IR-Strahler erkannt *)
    Data.UV1_Detected    := (Data.StatusByte AND 16#20) <> 16#00; (* Bit 5: 1 = UV-LED 1 erkannt *)
    Data.UV2_Detected    := (Data.StatusByte AND 16#10) <> 16#00; (* Bit 4: 1 = UV-LED 2 erkannt *)
    Data.IR_Level_OK     := (Data.StatusByte AND 16#08) = 16#00;  (* Bit 3: 0 = Normal > 50%, 1 = Fehler < 50% *)
    Data.UV1_Level_Error := (Data.StatusByte AND 16#02) <> 16#00; (* Bit 1: 1 = UV-LED 1 Pegelfehler *)
    Data.UV2_Level_Error := (Data.StatusByte AND 16#01) <> 16#00; (* Bit 0: 1 = UV-LED 2 Pegelfehler *)

    (* Fehlerbehandlung direkt aus den Statusbits des Sensors *)
    IF NOT Data.IR_Detected THEN
        Data.Error     := TRUE;
        Data.ErrorCode := MF_ERR_IR_LAMP_MISSING;
        Data.ErrorText := 'Gerätefehler: IR-Quelle nicht erkannt oder defekt';
    ELSIF NOT Data.IR_Level_OK THEN
        Data.Error     := TRUE;
        Data.ErrorCode := MF_ERR_IR_LAMP_LEVEL;
        Data.ErrorText := 'Gerätefehler: IR-Pegel < 50% (Verschmutzung oder Alterung)';
    ELSIF (Data.Gastype_CH1 = 'SO2' OR Data.Gastype_CH1 = 'NO' OR Data.Gastype_CH1 = 'NO2' OR Data.Gastype_CH1 = 'O3') AND Data.UV1_Level_Error THEN
        Data.Error     := TRUE;
        Data.ErrorCode := MF_ERR_UV_LEVEL;
        Data.ErrorText := 'Gerätefehler: UV-LED 1 Pegelfehler';
    ELSE
        (* Wenn kein Gerätefehler ansteht und kein Timeout aktiv ist -> OK *)
        IF Data.ErrorCode <> MF_ERR_COMM_TIMEOUT THEN
            Data.Error     := FALSE;
            Data.ErrorCode := MF_ERR_NONE;
            Data.ErrorText := 'OK';
        END_IF;
    END_IF;
END_IF;

(* ============================================================================ *)
(* Flankenauswertung für Sonderbefehle                                          *)
(* ============================================================================ *)
IF Cmd_ZeroCalibration AND NOT oldZeroCalib AND eState = MF_STATE_READY THEN
    eState  := MF_STATE_ZERO_CALIB;
    subStep := 0;
END_IF;
oldZeroCalib := Cmd_ZeroCalibration;

IF Cmd_ResetDevice AND NOT oldResetDev AND eState = MF_STATE_READY THEN
    eState  := MF_STATE_RESET_DEVICE;
    subStep := 0;
END_IF;
oldResetDev := Cmd_ResetDevice;

(* ============================================================================ *)
(* Zustandsmaschine (State Machine)                                            *)
(* ============================================================================ *)
Data.State := eState;

CASE eState OF

    (* ------------------------------------------------------------------------ *)
    (* DISABLED                                                                 *)
    (* ------------------------------------------------------------------------ *)
    MF_STATE_DISABLED:
        Data.StateText := 'Deaktiviert';
        IF Enable THEN
            eState := MF_STATE_INIT_START;
        END_IF;

    (* ------------------------------------------------------------------------ *)
    (* INIT_START                                                               *)
    (* ------------------------------------------------------------------------ *)
    MF_STATE_INIT_START:
        Data.StateText := 'Initialisiere...';
        subStep        := 0;
        timeoutCounter := 0;
        eState         := MF_STATE_READ_SN;

    (* ------------------------------------------------------------------------ *)
    (* 1. Seriennummer abfragen (Cmd 16#40)                                     *)
    (* ------------------------------------------------------------------------ *)
    MF_STATE_READ_SN:
        Data.StateText := 'Lese Seriennummer...';
        IF subStep = 0 THEN
            Bus.TxData[0] := 16#40; Bus.TxData[1] := 16#00; Bus.TxData[2] := 16#00; Bus.TxData[3] := 16#00;
            Bus.TxData[4] := 16#00; Bus.TxData[5] := 16#00; Bus.TxData[6] := 16#55; Bus.TxData[7] := 16#30;
            Bus.TxReq := TRUE;
            subStep   := 1;
        ELSIF subStep = 1 THEN
            tTimeout(IN := TRUE, PT := TimeoutTime);
            IF Bus.RxNew AND Bus.RxData[0] = 16#40 THEN
                tTimeout(IN := FALSE);
                Data.SerialNumber := WORD_TO_UINT(SHL(BYTE_TO_WORD(Bus.RxData[3]), 8) OR BYTE_TO_WORD(Bus.RxData[2]));
                subStep := 0;
                eState  := MF_STATE_READ_SW_REV;
            ELSIF tTimeout.Q THEN
                tTimeout(IN := FALSE);
                Data.Connected := FALSE;
                Data.Error     := TRUE;
                Data.ErrorCode := MF_ERR_COMM_TIMEOUT;
                Data.ErrorText := 'Timeout bei Abfrage Seriennummer';
                subStep := 0;
                eState  := MF_STATE_ERROR;
            END_IF;
        END_IF;

    (* ------------------------------------------------------------------------ *)
    (* 2. Firmware-Revision abfragen (Cmd 16#0B)                                *)
    (* ------------------------------------------------------------------------ *)
    MF_STATE_READ_SW_REV:
        Data.StateText := 'Lese Firmware-Version...';
        IF subStep = 0 THEN
            Bus.TxData[0] := 16#0B; Bus.TxData[1] := 16#00; Bus.TxData[2] := 16#00; Bus.TxData[3] := 16#00;
            Bus.TxData[4] := 16#00; Bus.TxData[5] := 16#00; Bus.TxData[6] := 16#55; Bus.TxData[7] := 16#30;
            Bus.TxReq := TRUE;
            subStep   := 1;
        ELSIF subStep = 1 THEN
            tTimeout(IN := TRUE, PT := TimeoutTime);
            IF Bus.RxNew AND Bus.RxData[0] = 16#0B THEN
                tTimeout(IN := FALSE);
                Data.SoftwareRevision := WORD_TO_UINT(SHL(BYTE_TO_WORD(Bus.RxData[3]), 8) OR BYTE_TO_WORD(Bus.RxData[2]));
                subStep := 0;
                eState  := MF_STATE_READ_CONFIG_ID;
            ELSIF tTimeout.Q THEN
                tTimeout(IN := FALSE);
                Data.Connected := FALSE;
                Data.Error     := TRUE;
                Data.ErrorCode := MF_ERR_COMM_TIMEOUT;
                Data.ErrorText := 'Timeout bei Abfrage Firmware';
                subStep := 0;
                eState  := MF_STATE_ERROR;
            END_IF;
        END_IF;

    (* ------------------------------------------------------------------------ *)
    (* 3. Config-ID & Gastyp abfragen (Cmd 16#62)                               *)
    (* ------------------------------------------------------------------------ *)
    MF_STATE_READ_CONFIG_ID:
        Data.StateText := 'Lese Gastyp (Config ID)...';
        IF subStep = 0 THEN
            Bus.TxData[0] := 16#62; Bus.TxData[1] := 16#00; Bus.TxData[2] := 16#00; Bus.TxData[3] := 16#00;
            Bus.TxData[4] := 16#00; Bus.TxData[5] := 16#00; Bus.TxData[6] := 16#55; Bus.TxData[7] := 16#30;
            Bus.TxReq := TRUE;
            subStep   := 1;
        ELSIF subStep = 1 THEN
            tTimeout(IN := TRUE, PT := TimeoutTime);
            IF Bus.RxNew AND Bus.RxData[0] = 16#62 THEN
                tTimeout(IN := FALSE);
                dwHelper := SHL(BYTE_TO_DWORD(Bus.RxData[5]), 24) OR SHL(BYTE_TO_DWORD(Bus.RxData[4]), 16) OR
                            SHL(BYTE_TO_DWORD(Bus.RxData[3]), 8)  OR BYTE_TO_DWORD(Bus.RxData[2]);
                Data.ConfigID := dwHelper;

                (* Gastyp für Kanal 1 (Nibble 3: Bits 12..15 laut Handbuch S. 10/11) *)
                nGasIdx := DWORD_TO_USINT(SHR(dwHelper, 12) AND 16#0F);
                CASE nGasIdx OF
                    0: Data.Gastype_CH1 := 'none';
                    1: Data.Gastype_CH1 := 'SO2';
                    2: Data.Gastype_CH1 := 'CO2';
                    3: Data.Gastype_CH1 := 'CO';
                    4: Data.Gastype_CH1 := 'NO';
                    5: Data.Gastype_CH1 := 'NO2';
                    6: Data.Gastype_CH1 := 'N2O';
                    7: Data.Gastype_CH1 := 'H2S';
                    8: Data.Gastype_CH1 := 'CH4';
                    9: Data.Gastype_CH1 := 'CnHm';
                    16#0A: Data.Gastype_CH1 := 'Cl2';
                    16#0B: Data.Gastype_CH1 := 'H2O';
                    16#0C: Data.Gastype_CH1 := 'ClO2';
                    16#0D: Data.Gastype_CH1 := 'O3';
                    16#0E: Data.Gastype_CH1 := 'SF6';
                    16#0F: Data.Gastype_CH1 := 'CF4';
                    ELSE   Data.Gastype_CH1 := 'Unknown';
                END_CASE;

                subStep := 0;
                eState  := MF_STATE_READ_RANGE;
            ELSIF tTimeout.Q THEN
                tTimeout(IN := FALSE);
                Data.Connected := FALSE;
                Data.Error     := TRUE;
                Data.ErrorCode := MF_ERR_COMM_TIMEOUT;
                Data.ErrorText := 'Timeout bei Abfrage Config-ID';
                subStep := 0;
                eState  := MF_STATE_ERROR;
            END_IF;
        END_IF;

    (* ------------------------------------------------------------------------ *)
    (* 4. Messbereichsendwert CH1 abfragen (Cmd 16#47, Index 16#02)              *)
    (* ------------------------------------------------------------------------ *)
    MF_STATE_READ_RANGE:
        Data.StateText := 'Lese Messbereichsendwert...';
        IF subStep = 0 THEN
            Bus.TxData[0] := 16#47; Bus.TxData[1] := 16#02; Bus.TxData[2] := 16#00; Bus.TxData[3] := 16#00;
            Bus.TxData[4] := 16#00; Bus.TxData[5] := 16#00; Bus.TxData[6] := 16#55; Bus.TxData[7] := 16#30;
            Bus.TxReq := TRUE;
            subStep   := 1;
        ELSIF subStep = 1 THEN
            tTimeout(IN := TRUE, PT := TimeoutTime);
            IF Bus.RxNew AND Bus.RxData[0] = 16#47 AND Bus.RxData[1] = 16#02 THEN
                tTimeout(IN := FALSE);
                dwHelper := SHL(BYTE_TO_DWORD(Bus.RxData[5]), 24) OR SHL(BYTE_TO_DWORD(Bus.RxData[4]), 16) OR
                            SHL(BYTE_TO_DWORD(Bus.RxData[3]), 8)  OR BYTE_TO_DWORD(Bus.RxData[2]);
                pRealHelper := ADR(dwHelper);
                Data.MeasurementRange_CH1 := pRealHelper^;
                subStep := 0;
                eState  := MF_STATE_READ_UNIT;
            ELSIF tTimeout.Q THEN
                tTimeout(IN := FALSE);
                Data.Connected := FALSE;
                Data.Error     := TRUE;
                Data.ErrorCode := MF_ERR_COMM_TIMEOUT;
                Data.ErrorText := 'Timeout bei Abfrage Messbereich';
                subStep := 0;
                eState  := MF_STATE_ERROR;
            END_IF;
        END_IF;

    (* ------------------------------------------------------------------------ *)
    (* 5. Messeinheit CH1 abfragen (Cmd 16#61, Index 16#02)                     *)
    (* ------------------------------------------------------------------------ *)
    MF_STATE_READ_UNIT:
        Data.StateText := 'Lese Messeinheit...';
        IF subStep = 0 THEN
            Bus.TxData[0] := 16#61; Bus.TxData[1] := 16#02; Bus.TxData[2] := 16#00; Bus.TxData[3] := 16#00;
            Bus.TxData[4] := 16#00; Bus.TxData[5] := 16#00; Bus.TxData[6] := 16#55; Bus.TxData[7] := 16#30;
            Bus.TxReq := TRUE;
            subStep   := 1;
        ELSIF subStep = 1 THEN
            tTimeout(IN := TRUE, PT := TimeoutTime);
            IF Bus.RxNew AND Bus.RxData[0] = 16#61 AND Bus.RxData[1] = 16#02 THEN
                tTimeout(IN := FALSE);
                nUnitVal := WORD_TO_UINT(SHL(BYTE_TO_WORD(Bus.RxData[3]), 8) OR BYTE_TO_WORD(Bus.RxData[2]));
                IF nUnitVal = 0 THEN
                    Data.MeasurementUnit_CH1 := 'ppm';
                ELSIF nUnitVal = 1 THEN
                    Data.MeasurementUnit_CH1 := 'Vol.%';
                ELSE
                    Data.MeasurementUnit_CH1 := 'Raw';
                END_IF;
                subStep := 0;
                eState  := MF_STATE_READ_OP_HOURS;
            ELSIF tTimeout.Q THEN
                tTimeout(IN := FALSE);
                Data.Connected := FALSE;
                Data.Error     := TRUE;
                Data.ErrorCode := MF_ERR_COMM_TIMEOUT;
                Data.ErrorText := 'Timeout bei Abfrage Messeinheit';
                subStep := 0;
                eState  := MF_STATE_ERROR;
            END_IF;
        END_IF;

    (* ------------------------------------------------------------------------ *)
    (* 6. Betriebsstunden abfragen (Cmd 16#43)                                  *)
    (* ------------------------------------------------------------------------ *)
    MF_STATE_READ_OP_HOURS:
        Data.StateText := 'Lese Betriebsstunden...';
        IF subStep = 0 THEN
            Bus.TxData[0] := 16#43; Bus.TxData[1] := 16#00; Bus.TxData[2] := 16#00; Bus.TxData[3] := 16#00;
            Bus.TxData[4] := 16#00; Bus.TxData[5] := 16#00; Bus.TxData[6] := 16#55; Bus.TxData[7] := 16#30;
            Bus.TxReq := TRUE;
            subStep   := 1;
        ELSIF subStep = 1 THEN
            tTimeout(IN := TRUE, PT := TimeoutTime);
            IF Bus.RxNew AND Bus.RxData[0] = 16#43 THEN
                tTimeout(IN := FALSE);
                Data.OperatingHours := WORD_TO_UINT(SHL(BYTE_TO_WORD(Bus.RxData[3]), 8) OR BYTE_TO_WORD(Bus.RxData[2]));

                (* Init erfolgreich abgeschlossen! *)
                Data.Connected := TRUE;
                Data.Error     := FALSE;
                Data.ErrorCode := MF_ERR_NONE;
                Data.ErrorText := 'OK';
                subStep        := 0;
                eState         := MF_STATE_READY;
            ELSIF tTimeout.Q THEN
                tTimeout(IN := FALSE);
                Data.Connected := FALSE;
                Data.Error     := TRUE;
                Data.ErrorCode := MF_ERR_COMM_TIMEOUT;
                Data.ErrorText := 'Timeout bei Abfrage Betriebsstunden';
                subStep := 0;
                eState  := MF_STATE_ERROR;
            END_IF;
        END_IF;

    (* ------------------------------------------------------------------------ *)
    (* READY: Bereit & zyklisches Polling                                       *)
    (* ------------------------------------------------------------------------ *)
    MF_STATE_READY:
        Data.StateText := 'Bereit / Messung aktiv';
        subStep        := 0;
        tTimeout(IN := FALSE);

        tPollConc(IN := NOT tPollConc.Q, PT := PollInterval_Conc);
        tPollTemp(IN := NOT tPollTemp.Q, PT := PollInterval_Temp);

        IF tPollConc.Q THEN
            queryCH2Active := FALSE;
            eState := MF_STATE_POLL_CONC;
        ELSIF tPollTemp.Q THEN
            eState := MF_STATE_POLL_TEMP;
        END_IF;

    (* ------------------------------------------------------------------------ *)
    (* POLL_CONC: Gaskonzentration abfragen                                     *)
    (* ------------------------------------------------------------------------ *)
    MF_STATE_POLL_CONC:
        Data.StateText := 'Messe Konzentration...';
        IF subStep = 0 THEN
            Bus.TxData[0] := 16#17;
            IF queryCH2Active THEN
                Bus.TxData[1] := 16#01; (* CH2 *)
            ELSE
                Bus.TxData[1] := 16#00; (* CH1 *)
            END_IF;
            Bus.TxData[2] := 16#00; Bus.TxData[3] := 16#00; Bus.TxData[4] := 16#00; Bus.TxData[5] := 16#00;
            Bus.TxData[6] := 16#55; Bus.TxData[7] := 16#30;
            Bus.TxReq := TRUE;
            subStep   := 1;

        ELSIF subStep = 1 THEN
            tTimeout(IN := TRUE, PT := TimeoutTime);

            IF Bus.RxNew AND Bus.RxData[0] = 16#17 THEN
                tTimeout(IN := FALSE);
                timeoutCounter := 0;
                Data.Connected := TRUE;

                dwHelper := SHL(BYTE_TO_DWORD(Bus.RxData[5]), 24) OR SHL(BYTE_TO_DWORD(Bus.RxData[4]), 16) OR
                            SHL(BYTE_TO_DWORD(Bus.RxData[3]), 8)  OR BYTE_TO_DWORD(Bus.RxData[2]);
                pRealHelper := ADR(dwHelper);

                IF Bus.RxData[1] = 16#00 THEN
                    Data.Concentration_CH1 := pRealHelper^;
                    IF ReadCH2 THEN
                        queryCH2Active := TRUE;
                        subStep        := 0; (* Direkt Kanal 2 abfragen *)
                    ELSE
                        eState         := MF_STATE_READY;
                    END_IF;
                ELSIF Bus.RxData[1] = 16#01 THEN
                    Data.Concentration_CH2 := pRealHelper^;
                    eState                 := MF_STATE_READY;
                END_IF;

            ELSIF tTimeout.Q THEN
                tTimeout(IN := FALSE);
                timeoutCounter := timeoutCounter + 1;
                IF timeoutCounter >= 3 THEN
                    Data.Connected := FALSE;
                    Data.Error     := TRUE;
                    Data.ErrorCode := MF_ERR_COMM_TIMEOUT;
                    Data.ErrorText := 'Kommunikations-Timeout (Keine Antwort)';
                    eState         := MF_STATE_ERROR;
                ELSE
                    eState := MF_STATE_READY;
                END_IF;
            END_IF;
        END_IF;

    (* ------------------------------------------------------------------------ *)
    (* POLL_TEMP: Detektortemperatur abfragen                                   *)
    (* ------------------------------------------------------------------------ *)
    MF_STATE_POLL_TEMP:
        Data.StateText := 'Messe Temperatur...';
        IF subStep = 0 THEN
            Bus.TxData[0] := 16#18; Bus.TxData[1] := 16#00; Bus.TxData[2] := 16#00; Bus.TxData[3] := 16#00;
            Bus.TxData[4] := 16#00; Bus.TxData[5] := 16#00; Bus.TxData[6] := 16#55; Bus.TxData[7] := 16#30;
            Bus.TxReq := TRUE;
            subStep   := 1;

        ELSIF subStep = 1 THEN
            tTimeout(IN := TRUE, PT := TimeoutTime);

            IF Bus.RxNew AND Bus.RxData[0] = 16#18 THEN
                tTimeout(IN := FALSE);
                timeoutCounter := 0;

                dwHelper := SHL(BYTE_TO_DWORD(Bus.RxData[5]), 24) OR SHL(BYTE_TO_DWORD(Bus.RxData[4]), 16) OR
                            SHL(BYTE_TO_DWORD(Bus.RxData[3]), 8)  OR BYTE_TO_DWORD(Bus.RxData[2]);
                pRealHelper := ADR(dwHelper);
                Data.Temperature_CH1 := pRealHelper^;
                eState := MF_STATE_READY;

            ELSIF tTimeout.Q THEN
                tTimeout(IN := FALSE);
                timeoutCounter := timeoutCounter + 1;
                IF timeoutCounter >= 3 THEN
                    Data.Connected := FALSE;
                    Data.Error     := TRUE;
                    Data.ErrorCode := MF_ERR_COMM_TIMEOUT;
                    Data.ErrorText := 'Kommunikations-Timeout (Keine Antwort)';
                    eState         := MF_STATE_ERROR;
                ELSE
                    eState := MF_STATE_READY;
                END_IF;
            END_IF;
        END_IF;

    (* ------------------------------------------------------------------------ *)
    (* ZERO_CALIB: Nullpunkt-Kalibrierung auslösen                              *)
    (* ------------------------------------------------------------------------ *)
    MF_STATE_ZERO_CALIB:
        Data.StateText := 'Nullpunkt-Kalibrierung...';
        IF subStep = 0 THEN
            Bus.TxData[0] := 16#11; Bus.TxData[1] := 16#00; Bus.TxData[2] := 16#00; Bus.TxData[3] := 16#00;
            Bus.TxData[4] := 16#00; Bus.TxData[5] := 16#00; Bus.TxData[6] := 16#55; Bus.TxData[7] := 16#30;
            Bus.TxReq := TRUE;
            subStep   := 1;
        ELSIF subStep = 1 THEN
            tTimeout(IN := TRUE, PT := T#500ms);
            IF Bus.RxNew AND Bus.RxData[0] = 16#11 THEN
                tTimeout(IN := FALSE);
                subStep := 0;
                eState  := MF_STATE_READY;
            ELSIF tTimeout.Q THEN
                tTimeout(IN := FALSE);
                subStep := 0;
                eState  := MF_STATE_READY;
            END_IF;
        END_IF;

    (* ------------------------------------------------------------------------ *)
    (* RESET_DEVICE: Sensor per Software neu starten                            *)
    (* ------------------------------------------------------------------------ *)
    MF_STATE_RESET_DEVICE:
        Data.StateText := 'Sensor wird neu gestartet...';
        IF subStep = 0 THEN
            Bus.TxData[0] := 16#04; Bus.TxData[1] := 16#00; Bus.TxData[2] := 16#00; Bus.TxData[3] := 16#00;
            Bus.TxData[4] := 16#00; Bus.TxData[5] := 16#00; Bus.TxData[6] := 16#55; Bus.TxData[7] := 16#30;
            Bus.TxReq := TRUE;
            subStep   := 1;
        ELSIF subStep = 1 THEN
            tTimeout(IN := TRUE, PT := T#1s);
            IF Bus.RxNew OR tTimeout.Q THEN
                tTimeout(IN := FALSE);
                subStep := 0;
                eState  := MF_STATE_INIT_START; (* Nach Reset komplett neu identifizieren *)
            END_IF;
        END_IF;

    (* ------------------------------------------------------------------------ *)
    (* ERROR                                                                    *)
    (* ------------------------------------------------------------------------ *)
    MF_STATE_ERROR:
        Data.StateText := 'Fehler';
        Data.Error     := TRUE;
        Bus.TxReq      := FALSE;
        IF Reset THEN
            Data.Error     := FALSE;
            Data.ErrorCode := MF_ERR_NONE;
            Data.ErrorText := 'OK';
            timeoutCounter := 0;
            subStep        := 0;
            eState         := MF_STATE_INIT_START;
        END_IF;

END_CASE;

END_FUNCTION_BLOCK

(* ---- FB_TaskManager.st ---- *)
FUNCTION_BLOCK FB_TaskManager
VAR_INPUT
	newOrder : STRING;
	response: BOOL;	(*Response from the serial connection*)
END_VAR

VAR_OUTPUT
	queued: BOOL;
	commandReady: BOOL := FALSE; (* Flag to indicate a command is ready to be sent *)
	currentOrder: STRING;
END_VAR

VAR
	orderQueue: ARRAY[1..100] OF STRING;
	queueHead: INT :=1;
	queueTail: INT :=1;
	orderInProgress: BOOL := FALSE;
(*	lastOrder : STRING := ''; *)
END_VAR

(*	IF lastOrder <> newOrder THEN *)
(*		Act_AddOrder; *)
(*	END_IF *)
	;
END_FUNCTION_BLOCK

ACTIONS

	ACTION Act_AddOrder
		IF (queueTail MOD 100) + 1 <> queueHead THEN
			(* IF newOrder <> orderQueue[queueTail-1] THEN (* reject command if already exists *) *)
				orderQueue[queueTail] := newOrder;
				queueTail := (queueTail MOD 100) + 1;
				queued := TRUE;
	(*			lastOrder := newOrder; *)
			(* END_IF *)
		ELSE
			queued := FALSE; (* success: BOOL; *)
		END_IF
	END_ACTION

	ACTION Act_ProcessOrder

		IF NOT orderInProgress AND queueHead <> queueTail THEN
			currentOrder := orderQueue[queueHead];
			queueHead := (queueHead MOD 100) + 1;
			orderInProgress := TRUE;
			commandReady := TRUE; (* Set the flag to indicate the command is ready *)
		END_IF

		IF response THEN (*Reset the flags*)
			orderInProgress := FALSE;
			commandReady := FALSE;
			response := FALSE;
		END_IF

	END_ACTION

END_ACTIONS
